# B&R Automation Studio project AriesV2 (part 2)

### _X_bgftpclient.c
```c
#include <bur/plc.h>
#include <bur/plctypes.h>
#include <ethernet.h>
#include <ethsock.h>
#include <asstring.h>
#include <brsystem.h>
#include <sys_lib.h>

#include "bgsprintf.h"
#include "bgstatemachine.h"
#include "bgstring.h"
#include "bgFtpClient.h"

#include "bgdebug.h"

#include "bgstatemachine.c"
#include "bgsprintf.c"
#include "bgstring.c"

/*
History:
9/11/2005
- added support for receiving large files over ftp
- added error event for user ftp commands:
int bgFtpClientCmd<CmdName>OnError(bgFtpClient_typ *p);

*/

void ftpClientConnect(bgFtpClient_typ *p, int msgId);
int ftpClientConnectOnDone(bgFtpClient_typ *p);
int ftpClientConnectOnError(bgFtpClient_typ *p);

void ftpClientLogin(bgFtpClient_typ *p, int msgId);
int ftpClientLoginOnDone(bgFtpClient_typ *p);
int ftpClientLoginOnError(bgFtpClient_typ *p);

void ftpClientLogout(bgFtpClient_typ *p, int msgId);
int ftpClientLogoutOnDone(bgFtpClient_typ *p);
int ftpClientLogoutOnError(bgFtpClient_typ *p);

void ftpClientCmdGetFile(bgFtpClient_typ *p);

void ftpClientCmdList(bgFtpClient_typ *p);

void ftpClientCmdPwd(bgFtpClient_typ *p);

void ftpClientCmdCwd(bgFtpClient_typ *p);

void ftpClientDataServer(bgFtpClient_typ *p, int msgId);
int ftpClientDataServerOnError(bgFtpClient_typ *p);
int ftpClientDataServerOnDone(bgFtpClient_typ *p);

void ftpClientSingleCmdInit(bgFtpClient_typ *p, char *cmd, char *expectedServerResponse);
void ftpClientSingleCmd(bgFtpClient_typ *p);
int ftpClientSingleCmdOnError(bgFtpClient_typ *p);
int ftpClientSingleCmdOnDone(bgFtpClient_typ *p);

void ftpClientExecuteUserCmd_cyclic(bgFtpClient_typ *p);

int ftpClientCmdMultiOnDone(bgFtpClient_typ *p, int cmdId);
int ftpClientMultiCmdOnError(bgFtpClient_typ *p, int cmdId);
int ftpClientCmdCheckServerResponseCode(bgFtpClient_typ *p);

void ftpClientInitDataPort(bgFtpClient_typ *p);
void swapBytesInShort(unsigned short *value);
void setSocketAddressData(ETH_sockaddr_typ *adrData, char *hostIpAddressString, unsigned short hostPort);
void ftpClientGetResponse(bgFtpClient_typ *p);

void ftpClientCmdTextPort(bgFtpClient_typ *p, char *textBuffer);
void ftpClientMutliStateCmdErrorLog(bgFtpClient_typ *p);

int ftpClientIncrDataPort(bgFtpClient_typ *p);

/*
########################################################################################
========================================================================================
- FTP client protocol main state machine
- must be executed as a cyclic task (<=100ms)
- protocol implemenation uses nested state machines (several levels deep)
- FTP functions such as: connect, disconnect, login, logout and different FTP commands
are all implemented as state machines
*/
void bgFtpClientCyclic(bgFtpClient_typ *p, int msgId)
{
bgStateMachine_typ *psm = &p->smFtp;

	/*FTP client top level state machine*/
	switch( bgSMCyclic(psm) ){
		case 1:
          	/*idle; monitor user connection request flag*/
			bgSMSetStateName(psm, "Idle");

          	if(p->user.connectRequest){
	            p->user.connectRequest = 0;
	            p->user.disconnectRequest = 0;
				bgSMSetNextState(psm, bgSMGetState(psm) + 1);
          	}
		break;
		case 2:
			/*connect to FTP server*/
			bgSMSetStateName(psm, "Connect");

			if(bgSMIsStateInit(psm)){
				ftpClientConnect(p, BGSM_MSGID_INIT);
			}

			ftpClientConnect(p, BGSM_MSGID_CYCLIC);

			/*check if we are connected to FTP server*/
			if( p->isConnected ){
				bgSMSetNextState(psm, bgSMGetState(psm) + 1);
			}

			if(	ftpClientConnectOnError(p)){
                ERRxwarning(USER_ERROR_FTP, 1, "ftpClient-Err-socket()");
				bgSMRaiseError(psm, "error in lower level SM", 1, 0);
            }
		break;
		case 3:
			/*login*/
			bgSMSetStateName(psm, "Login");

			if(bgSMIsStateInit(psm)){
				ftpClientLogin(p, BGSM_MSGID_INIT);
			}

			ftpClientLogin(p, BGSM_MSGID_CYCLIC);

			/*check if we are looged-in*/
			if(p->isLoggedIn){
				p->userState = 0;
				bgSMSetNextState(psm, bgSMGetState(psm) + 1);
			}
			if(ftpClientLoginOnError(p)){
                ERRxwarning(USER_ERROR_FTP, 1, "ftpClient-Err-login()");
				bgSMRaiseError(psm, "error in lower level SM", 0, 0);
            }
		break;
		case 4:
            /*connected & logged-in -> normal operational state*/
			bgSMSetStateName(psm, "Ready");

			/*monitor requests & execute FTP commands*/
			ftpClientExecuteUserCmd_cyclic(p);

			/*terminate if socket error detected*/
			if(p->cmdError == ERR_SOCKET){
				bgSMSetNextState(psm, bgSMGetState(psm) + 1);
			}

			if(p->test){
				p->test = 0;
				ftpClientGetResponse(p);
			}

            /*monitor user disconnect request*/
            /*NOTE: upon receiving request, make sure to wait that FTP command in progress completes!*/

			/*disconnect allowed only after command completes*/
            if(p->user.disconnectRequest && !p->userState){
                p->user.connectRequest = 0;
                p->user.disconnectRequest = 0;
				bgSMSetNextState(psm, bgSMGetState(psm) + 1);
            }
		break;
		case 5:
            /*logout*/
			bgSMSetStateName(psm, "Logout");

			if(bgSMIsStateInit(psm)){
				ftpClientLogout(p, BGSM_MSGID_INIT);
			}

			ftpClientLogout(p, BGSM_MSGID_CYCLIC);

			/*chech if we are logged out*/
			if(!p->isLoggedIn){
				bgSMSetNextState(psm, bgSMGetState(psm) + 1);
			}

			if(ftpClientLogoutOnError(p)){
                ERRxwarning(USER_ERROR_FTP, 1, "ftpClient-Err-socket()");
				bgSMRaiseError(psm, "error in lower level SM", 0, 0);
            }
		break;
		case 6:
			bgSMSetStateName(psm, "Close CMD socket");
            /*normal operation; close socket*/
			bgSMRaiseDone(psm, 0);
		break;
		default:
			/*unhandled state*/
			bgSMRaiseError(psm, "unknown state", 0, bgSMGetState(psm));
		break;
	}

	if(bgSMOnDone(psm)){
		/*error state; socket closing is needed*/
		close(p->sock);

		p->isConnected = 0;

		bgSMSetNextState(psm, 1);
	}

	if(bgSMOnError(psm)){
		/*check if socket close needed or not?*/
		if( !bgSMGetErrorId(psm) )
			close(p->sock);

		p->isConnected = 0;
		p->cmdError = 1;
		bgSMSetNextState(psm, 1);
	}
}
/*
########################################################################################
	 INDIVIDUAL FTP COMMANDS
- each individual FTP command has following USER level interface methods:
	ftpClientCmd<Name>Init()
		- start command execution; pass-in user parameters; init cmd state machine
	ftpClientCmd<Name>OnDone()
		- monitor cmd completion (0-not complete; 1-complete)

- each command also has core implemenation (not used or called by the user)
	ftpClientCmd<Name>()

- FTP commands such as: PWD, CWD, PUT, GET, DIR are multi-level commands: it usually takes
several primitive FTP commands (i.e. PORT, TYPE, RETR etc) to complete one FTP command

########################################################################################
*/

/*
========================================================================================
- state machine that handles execution of individual, multi-level FTP commands
- FTP client executes one Multi-level command at the time
*/
void ftpClientExecuteUserCmd_cyclic(bgFtpClient_typ *p)
{
	/*execute user commands*/
	switch(p->userState){
	/*idle*/
        case 0:
        break;
        case 1:
        break;
        case 2:
            ftpClientCmdList(p);
        break;
        case 4:
            ftpClientCmdPwd(p);
        break;
        case 6:
            ftpClientCmdGetFile(p);
        break;
        case 8:
            ftpClientCmdCwd(p);
        break;
        default:
            p->userState = 0;
        break;
	}

}

/*
========================================================================================
FTP Command Implementation:
GetFile
*/
void bgFtpClientCmdGetFileInit(bgFtpClient_typ *p, char *fileName, char* buffer, int bufferLength)
{
    /*select command to execute*/
	p->userState = 6;

	/*pass command parameters*/
	p->user.dataBuffer = buffer;
	p->user.dataBufferLength = bufferLength;
	strcpy(&p->user.fileName[0], fileName);

    /*start command execution*/
	bgSMReset(&p->smFtpMultiCmd);
}

int bgFtpClientCmdGetFileOnDone(bgFtpClient_typ *p)
{
	return ftpClientCmdMultiOnDone(p, 6);
}

int bgFtpClientCmdGetFileOnError(bgFtpClient_typ *p)
{
	return ftpClientMultiCmdOnError(p, 6);
}

void ftpClientCmdGetFile(bgFtpClient_typ *p)
{
char cmdText[256];
bgStateMachine_typ *psm = &p->smFtpMultiCmd;

	/*FTP client multi level command state machine*/
	switch( bgSMCyclic(psm) ){
		case 1:
          	/*idle - monitor user connection request flag*/
			bgSMSetStateName(psm, "GetFile-InitDataSocket");

			if( bgSMIsStateInit(psm) ){
				/*generate port number to use*/
				ftpClientIncrDataPort(p);
				/*init Data transport socket*/
	            ftpClientDataServer(p, BGSM_MSGID_INIT);
			}

			/*wait for ready msg from the DataServer*/
            if( p->isDataPortReady ){
				bgSMSetNextState(psm, bgSMGetState(psm) + 1);
            }
/*TODO: timeout*/
		break;
		case 2:
    		/*PORT command: "PORT 192,168,1,6,0,20<CR><LF>"*/
			bgSMSetStateName(psm, "GetFile-PORT");
			if(bgSMIsStateInit(psm)){
	    		/*send command*/
	            ftpClientCmdTextPort(p, &cmdText[0]);

	    		ftpClientSingleCmdInit(p, &cmdText[0], "2??");
			}

    		/*recv cmd response*/
    		ftpClientSingleCmd(p);
			if(ftpClientSingleCmdOnDone(p)){
				bgSMSetNextState(psm, bgSMGetState(psm) + 1);
			}
			if(ftpClientSingleCmdOnError(p)){
				bgSMRaiseError(psm, "error in lower level SM", 0, 0);
			}
		break;
		case 3:
    		/*TYPE command: "TYPE I<CR><LF>"*/
			bgSMSetStateName(psm, "GetFile-TYPE");
			if(bgSMIsStateInit(psm)){
	    		/*send command*/
	    		ftpClientSingleCmdInit(p, "TYPE I", "2??");
			}

    		/*recv cmd response*/
    		ftpClientSingleCmd(p);
			if(ftpClientSingleCmdOnDone(p)){
				bgSMSetNextState(psm, bgSMGetState(psm) + 1);
			}

			if(ftpClientSingleCmdOnError(p)){
				bgSMRaiseError(psm, "error in lower level SM", 0, 0);
			}
		break;
		case 4:
    		/*RETR command: "RETR<CR><LF>""*/
			bgSMSetStateName(psm, "GetFile-RETR");
			if(bgSMIsStateInit(psm)){
	    		/*send command*/
	    		/*send command*/
	    		strcpy(&cmdText[0], "RETR ");
	    		strcat(&cmdText[0], &p->user.fileName[0]);
	    		ftpClientSingleCmdInit(p, &cmdText[0], "2??");
			}

    		/*recv cmd response*/
    		ftpClientSingleCmd(p);
			if(ftpClientSingleCmdOnDone(p)){
				/*notify data port server that the response is comming*/
				ftpClientDataServer(p, 2);
				bgSMSetNextState(psm, bgSMGetState(psm) + 1);
			}

			if(ftpClientSingleCmdOnError(p)){
				bgSMRaiseError(psm, "error in lower level SM", 0, 0);
				/*close data server port*/
				ftpClientDataServer(p, 3);
			}
		break;
        case 5:
			bgSMSetStateName(psm, "GetFile-DATASRVR active");
        break;
		default:
			/*unhandled state*/
			bgSMRaiseError(psm, "unknown state", 0, bgSMGetState(psm));
		break;
	}

	if(bgSMOnError(psm)){
		p->isErrorMultiCmd = p->userState;
		p->userState = 0;
		return;
	}

	ftpClientDataServer(p, BGSM_MSGID_CYCLIC);

	if(ftpClientDataServerOnDone(p)){
		p->isDoneMultiCmd = p->userState;
		p->userState = 0;
	}

	if(ftpClientDataServerOnError(p)){
		p->isErrorMultiCmd = p->userState;
		p->userState = 0;
	}

}
/*
========================================================================================
FTP Command Implementation:
List (dir)
*/
void bgFtpClientCmdListInit(bgFtpClient_typ *p, char *buffer, int bufferLength)
{
    /*select command to execute*/
	p->userState = 2;

	/*pass command parameters*/
	p->user.dataBuffer = buffer;
	p->user.dataBufferLength = bufferLength;

    /*start command execution*/
	bgSMReset(&p->smFtpMultiCmd);
}

int bgFtpClientCmdListOnDone(bgFtpClient_typ *p)
{
	return ftpClientCmdMultiOnDone(p, 2);
}

int bgFtpClientCmdListOnError(bgFtpClient_typ *p)
{
	return ftpClientMultiCmdOnError(p, 2);

}

void ftpClientCmdList(bgFtpClient_typ *p)
{
char cmdText[64];
bgStateMachine_typ *psm = &p->smFtpMultiCmd;

	/*FTP client multi level command state machine*/
	switch( bgSMCyclic(psm) ){
		case 1:
          	/*idle - monitor user connection request flag*/
			bgSMSetStateName(psm, "List-InitDataSocket");

			if( bgSMIsStateInit(psm) ){
				/*generate port number to use*/
				ftpClientIncrDataPort(p);
				/*init Data transport socket*/
	            ftpClientDataServer(p, BGSM_MSGID_INIT);
			}

			/*wait for ready msg from the DataServer*/
            if( p->isDataPortReady ){
				bgSMSetNextState(psm, bgSMGetState(psm) + 1);
            }
/*TODO: timeout*/
		break;
		case 2:
    		/*PORT command: "PORT 192,168,1,6,0,20<CR><LF>"*/
			bgSMSetStateName(psm, "List-PORT");
			if(bgSMIsStateInit(psm)){
	    		/*send command*/
	            ftpClientCmdTextPort(p, &cmdText[0]);

	    		ftpClientSingleCmdInit(p, &cmdText[0], "2??");
			}

    		/*recv cmd response*/
    		ftpClientSingleCmd(p);
			if(ftpClientSingleCmdOnDone(p)){
				bgSMSetNextState(psm, bgSMGetState(psm) + 1);
			}
			if(ftpClientSingleCmdOnError(p)){
				bgSMRaiseError(psm, "error in lower level SM", 0, 0);
			}
		break;
		case 3:
    		/*TYPE command: "TYPE I<CR><LF>"*/
			bgSMSetStateName(psm, "List-TYPE");
			if(bgSMIsStateInit(psm)){
	    		/*send command*/
	    		ftpClientSingleCmdInit(p, "TYPE I", "2??");
			}

    		/*recv cmd response*/
    		ftpClientSingleCmd(p);
			if(ftpClientSingleCmdOnDone(p)){
				bgSMSetNextState(psm, bgSMGetState(psm) + 1);
			}

			if(ftpClientSingleCmdOnError(p)){
				bgSMRaiseError(psm, "error in lower level SM", 0, 0);
			}
		break;
		case 4:
    		/*LIST command: "LIST<CR><LF>""*/
			bgSMSetStateName(psm, "List-List");
			if(bgSMIsStateInit(psm)){
	    		/*send command*/
	    		ftpClientSingleCmdInit(p, "LIST", "2??");
			}

    		/*recv cmd response*/
    		ftpClientSingleCmd(p);
			if(ftpClientSingleCmdOnDone(p)){
				/*notify data port server that the response is comming*/
				ftpClientDataServer(p, 2);
				bgSMSetNextState(psm, bgSMGetState(psm) + 1);
			}

			if(ftpClientSingleCmdOnError(p)){
				/*close data server port*/
				ftpClientDataServer(p, 3);
				bgSMRaiseError(psm, "error in lower level SM", 0, 0);
			}
		break;
        case 5:
			bgSMSetStateName(psm, "List-DATASRVR active");
        break;
		default:
			/*unhandled state*/
			bgSMRaiseError(psm, "unknown state", 0, bgSMGetState(psm));
		break;
	}

	if(bgSMOnError(psm)){
		p->isErrorMultiCmd = p->userState;
		p->userState = 0;
		return;
	}

	ftpClientDataServer(p, BGSM_MSGID_CYCLIC);

	if(ftpClientDataServerOnDone(p)){
		p->isDoneMultiCmd = p->userState;
		p->userState = 0;
	}

	if(ftpClientDataServerOnError(p)){
		p->isErrorMultiCmd = p->userState;
		p->userState = 0;
	}
}
/*
========================================================================================
FTP Command Implementation:
Pwd (Print Working Directory)
*/
void bgFtpClientCmdPwdInit(bgFtpClient_typ *p, char *buffer, int bufferLength)
{
    /*select command to execute*/
	p->userState = 4;

	/*pass command parameters*/
	p->user.dataBuffer = buffer;
	p->user.dataBufferLength = bufferLength;

    /*start command execution*/
	bgSMReset(&p->smFtpMultiCmd);
}

int bgFtpClientCmdPwdOnDone(bgFtpClient_typ *p)
{
	return ftpClientCmdMultiOnDone(p, 4);
}

int bgFtpClientCmdPwdOnError(bgFtpClient_typ *p)
{
	return ftpClientMultiCmdOnError(p, 4);

}

void ftpClientCmdPwd(bgFtpClient_typ *p)
{
bgStateMachine_typ *psm = &p->smFtpMultiCmd;

	/*FTP client multi level command state machine*/
	switch( bgSMCyclic(psm) ){
		case 1:
    		/*XPWD command: "XPWD<CR><LF>"*/
			bgSMSetStateName(psm, "PWD");
			if(bgSMIsStateInit(psm)){
	    		/*send command*/
	    		ftpClientSingleCmdInit(p, "PWD", "2??");
			}

    		/*recv cmd response*/
    		ftpClientSingleCmd(p);

			if(ftpClientSingleCmdOnDone(p)){
				/*copy response strig into the user supplied buffer*/
				strcpy(p->user.dataBuffer, p->responseList.items[0]);
				bgSMRaiseDone(psm, 0);
			}

			if(ftpClientSingleCmdOnError(p)){
				bgSMRaiseError(psm, "got lower SM error", 0, 0);
			}
		break;
		default:
			/*unhandled state*/
			bgSMRaiseError(psm, "unknown state", 0, bgSMGetState(psm));
		break;
	}

	if(bgSMOnError(psm)){
		p->userState = 0;
	}

	if(bgSMOnDone(psm)){
		p->isDoneMultiCmd = p->userState;
		p->userState = 0;
	}

}
/*
========================================================================================
FTP Command Implementation:
Cwd (Change Working Directory)
*/
void bgFtpClientCmdCwdInit(bgFtpClient_typ *p, char *fileName, char *buffer, int bufferLength)
{
    /*select command to execute*/
	p->userState = 8;

	/*pass command parameters*/
	p->user.dataBuffer = buffer;
	p->user.dataBufferLength = bufferLength;
	strcpy(&p->user.fileName[0], fileName);

    /*start command execution*/
	bgSMReset(&p->smFtpMultiCmd);

}

int bgFtpClientCmdCwdOnDone(bgFtpClient_typ *p)
{
	return ftpClientCmdMultiOnDone(p, 8);
}

int bgFtpClientCmdCwdOnError(bgFtpClient_typ *p)
{
	return ftpClientMultiCmdOnError(p, 8);

}

void ftpClientCmdCwd(bgFtpClient_typ *p)
{
char cmdText[255];

bgStateMachine_typ *psm = &p->smFtpMultiCmd;

	/*FTP client multi level command state machine*/
	switch( bgSMCyclic(psm) ){
		case 1:
    		/*XPWD command: "CWD <fileName><CR><LF>"*/
			bgSMSetStateName(psm, "CWD");
			if(bgSMIsStateInit(psm)){
	    		/*send command: "CWD <fileName><CR><LF>"*/
	    		strcpy(&cmdText[0], "CWD ");
	    		strcat(&cmdText[0], &p->user.fileName[0]);
	    		ftpClientSingleCmdInit(p, &cmdText[0], "2??");
			}

    		/*recv cmd response*/
    		ftpClientSingleCmd(p);

			if(ftpClientSingleCmdOnDone(p)){
				/*copy response strig into the user supplied buffer*/
				strcpy(p->user.dataBuffer, p->responseList.items[0]);
				bgSMRaiseDone(psm, 0);
			}

			if(ftpClientSingleCmdOnError(p)){
				bgSMRaiseError(psm, "got lower SM error", 0, 0);
			}
		break;
	}

	if(bgSMOnError(psm)){
		p->isErrorMultiCmd = p->userState;
		p->userState = 0;
		return;
	}

	if(bgSMOnDone(psm)){
		p->isDoneMultiCmd = p->userState;
		p->userState = 0;
	}
}
/*
########################################################################################
========================================================================================
FTP Connect command state machine:
*/
int ftpClientConnectOnDone(bgFtpClient_typ *p){
	return bgSMOnDone(&p->smCmdSocket);
}

int ftpClientConnectOnError(bgFtpClient_typ *p){
	return bgSMOnError(&p->smCmdSocket);
}

void ftpClientConnect(bgFtpClient_typ *p, int msgId)
{
DINT ret;
bgStateMachine_typ *psm = & p->smCmdSocket;

	if( msgId == BGSM_MSGID_INIT){
		bgSMReset(psm);
	}

    switch(bgSMCyclic(psm)){
        case 1:
			bgSMSetStateName(psm, "Connect-CreateSocket");

			if( bgSMIsStateInit(psm) ){
				p->cmdError = 0;
				p->cmdErrorCode = 0;
				p->isConnected = 0;
				/*create socket*/
				p->sock = socket(ETH_AF_INET, ETH_SOCK_STREAM, 0);

				if( p->sock == ERR_SOCKET ){
					bgSMRaiseError(psm, "socket create err", 0, EthGetError());
					break;
				}

				/*set non-blocking socket operation*/
				{
					UDINT arg = 1;
					ioctl(p->sock, ETH_FIONBIO, (UDINT)&arg);
				}

				/*reset select flags*/
				fd_zero((UDINT)&p->fdR);
				fd_zero((UDINT)&p->fdW);

				/*set time-out to 10ms*/
				p->timeOut.tv_sec = 0;
				p->timeOut.tv_usec = 1000 * 10;

				/*adjust my own timeout counters*/
				p->sockData_TimerCounter = 0;
				p->sockData_TimerTime = 10;
#if 0
/*bind not necessary*/
				/*bind client socket*/
				ret = bind(p->sock, (UDINT)&p->ftpClientAdrData, sizeof(p->ftpClientAdrData));
				if(ret == ERR_SOCKET){
					bgSMRaiseError(psm, "socket bind err", 0, EthGetError());
					break;
				}
#endif
			}

			/*connect to remote host*/
			ret = connect(p->sock, (UDINT)&p->ftpServerAdrCmd, sizeof(p->ftpServerAdrCmd) );

			if(ret == ERR_SOCKET){
				UINT errCode = EthGetError();
				if(errCode == ERR_ETH_INPROGRESS){
					/*next: wait connect to complete*/
					bgSMSetNextState(psm, bgSMGetState(psm) + 1);
				    break;
				}else
				if(errCode == ERR_ETH_ISCONN){
					/*it's connected -> done*/
					ERRxwarning(USER_ERROR_FTP, errCode, "connect()-alreadyOK!");
					bgSMRaiseDone(psm, 0);
					break;
				}
				else{
					bgSMRaiseError(psm, "socket connect err", 0, EthGetError());
					break;
				}
			}
			/*connected!*/
			ERRxwarning(USER_ERROR_FTP, ret, "connect()-OK-Quick!");
			bgSMRaiseDone(psm, 0);
		break;
		case 2:
			bgSMSetStateName(psm, "Connect-Connect");

			/*select waits for connection to complete*/
			fd_set(p->sock, (UDINT)&p->fdR);
			fd_set(p->sock, (UDINT)&p->fdW);
			ret = sock_select(32, (UDINT)&p->fdR, (UDINT)&p->fdW, 0L, (UDINT)&p->timeOut);

			if(ret == ERR_SOCKET){
				bgSMRaiseError(psm, "socket connect err", 0, EthGetError());
				break;
			}
/*
			DBG("connect: ret=%d, error=%d\n\r", ret, EthGetError());
*/
			if(ret == 0){
				if( p->sockData_TimerCounter >= p->sockData_TimerTime ){
					/*NOTES:
					- trying to figure out how does the select timeout works in B&R!
					- using EthGetError() here is not needed, just to see what comes back
					*/
					bgSMRaiseError(psm, "connect timeout", 0, EthGetError());
				}else{
					p->sockData_TimerCounter++;
				}
			}else{
				if( fd_isset(p->sock, (UDINT)&p->fdW) ){
					bgSMRaiseDone(psm, 0);
				}
			}
		break;
		default:
			/*unhandled state*/
			bgSMRaiseError(psm, "unknown state", 0, bgSMGetState(psm));
		break;
    }

	if( bgSMOnDone(psm)){
		ERRxwarning(USER_ERROR_FTP, 0, "connect()-OK!");
		p->isConnected = 1;
	}

	if( bgSMOnError(psm)){

	}
}
/*
========================================================================================
*/
void ftpClientMutliStateCmdErrorLog(bgFtpClient_typ *p){
char text[64];
	/*log error*/
	strcpy(&text[0], "Err: ");
	strcat(&text[0], &p->cmdSendBuf[0]);
    ERRxwarning(USER_ERROR_FTP, p->cmdErrorCode, &text[0]);
}
/*
########################################################################################
========================================================================================
FTP Login command state machine:
-return values:
*/
int ftpClientLoginOnDone(bgFtpClient_typ *p){
	return bgSMOnDone(&p->smFtpMultiCmd);
}

int ftpClientLoginOnError(bgFtpClient_typ *p){
	return bgSMOnError(&p->smFtpMultiCmd);
}
void ftpClientLogin(bgFtpClient_typ *p, int msgId)
{
bgStateMachine_typ *psm = &p->smFtpMultiCmd;

	if( msgId == BGSM_MSGID_INIT){
		bgSMReset(psm);
	}

    switch(bgSMCyclic(psm)){
        case 1:
			/*send USER name*/
			bgSMSetStateName(psm, "Login-Welcome");

			if( bgSMIsStateInit(psm) ){
				/*send request*/
				/*ftpClientSingleCmdInit(p, 0, ">name");*/
				ftpClientSingleCmdInit(p, 0, ">FTP");
			}

			/*recv response*/
			ftpClientSingleCmd(p);

			if(ftpClientSingleCmdOnDone(p)){
				bgSMSetNextState(psm, bgSMGetState(psm) + 1);
			}

			if(ftpClientSingleCmdOnError(p)){
				bgSMRaiseError(psm, "error in lower level SM", 0, 0);
			}
        break;
        case 2:
			/*send USER name*/
			bgSMSetStateName(psm, "Login-UserName");

			if( bgSMIsStateInit(psm) ){
				/*send request*/
				ftpClientSingleCmdInit(p, "USER  anonymous", "331");
			}

			/*recv response*/
			ftpClientSingleCmd(p);

			if(ftpClientSingleCmdOnDone(p)){
				bgSMSetNextState(psm, bgSMGetState(psm) + 1);
			}

			if(ftpClientSingleCmdOnError(p)){
				bgSMRaiseError(psm, "error in lower level SM", 0, 0);
			}
        break;
        case 3:
			/*send PASSWORD */
			bgSMSetStateName(psm, "Login-Password");

			if( bgSMIsStateInit(psm) ){
				/*send request*/
				ftpClientSingleCmdInit(p, "PASS  anonymous@", "230");
			}

			/*recv response*/
			ftpClientSingleCmd(p);

			if(ftpClientSingleCmdOnDone(p)){
				bgSMRaiseDone(psm, 0);
			}

			if(ftpClientSingleCmdOnError(p)){
				bgSMRaiseError(psm, "error in lower level SM", 0, 0);
			}
        break;
        default:
			/*unhandled state*/
			bgSMRaiseError(psm, "unknown state", 0, bgSMGetState(psm));
        break;
    }

	if( bgSMOnDone(psm) ){
		p->isLoggedIn = 1;
	}

	if( bgSMOnError(psm) ){
		ftpClientMutliStateCmdErrorLog(p);
	}

}
/*
########################################################################################
========================================================================================
FTP Logout command state machine:
-return values:
*/
int ftpClientLogoutOnDone(bgFtpClient_typ *p){
	return bgSMOnDone(&p->smFtpMultiCmd);
}

int ftpClientLogoutOnError(bgFtpClient_typ *p){
	return bgSMOnError(&p->smFtpMultiCmd);
}

void ftpClientLogout(bgFtpClient_typ *p, int msgId)
{
bgStateMachine_typ *psm = &p->smFtpMultiCmd;

	if( msgId == BGSM_MSGID_INIT){
		bgSMReset(psm);
	}

    switch(bgSMCyclic(psm)){
        case 1:
			/*send USER name*/
			bgSMSetStateName(psm, "Logout-Quit");

			if( bgSMIsStateInit(psm) ){
				/*send request*/
				ftpClientSingleCmdInit(p, "QUIT", "2??");
			}

			/*recv response*/
			ftpClientSingleCmd(p);

			if(ftpClientSingleCmdOnDone(p)){
				bgSMRaiseDone(psm, 0);
			}

			if(ftpClientSingleCmdOnError(p)){
				bgSMRaiseError(psm, "error in lower level SM", 0, 0);
			}
        break;
        default:
			/*unhandled state*/
			bgSMRaiseError(psm, "unknown state", 0, bgSMGetState(psm));
        break;
    }

	if(bgSMOnDone(psm)){
		p->isLoggedIn = 0;
	}

	if(bgSMOnError(psm)){
		p->isLoggedIn = 0;
		ftpClientMutliStateCmdErrorLog(p);
	}
}
/*
########################################################################################
========================================================================================
Lowest level state machine handles execution of a single FTP request/response messaging

ftpClientSingleCmdInit();
	- selects command to execute; init command state machine

ftpClientSingleCmd();
	- command execution state machine

ftpClientCmdCheckServerResponseCode()
	- command response check and verification

*/
void ftpClientSingleCmdInit(bgFtpClient_typ *p, char *cmd, char *expectedServerResponse){
int i;

	/*copy command string into send buffer*/
	p->cmdSendBuf[0]=0;
	if(cmd){
		strcpy(&p->cmdSendBuf[0], cmd);
		/*append string termination -> CRLF*/
		strcat(&p->cmdSendBuf[0], "\r\n");
	}

	/*define expected server response string?*/
	p->cmdExpectedServerResponse[0] = 0;	/*don't care*/
	if(expectedServerResponse){
		/*is expected server response code or string?*/
		if( *expectedServerResponse == '>'){
			i = 1;
			p->cmdExpectedServerResponseCodeOrString = 1;	/*string*/
		}else{
			i = 0;
			p->cmdExpectedServerResponseCodeOrString = 0;	/*code*/
		}
		bgStrCpyN(&p->cmdExpectedServerResponse[0], expectedServerResponse+i, FTPCLIENT_RESPONSECODE_LEN);
	}

	/*clr rcv buffer string*/
	memset(&p->cmdRecvBuf[0], 0, FTPCLIENT_CMDBUFSIZE);
#if 0
/*clear response lines*/
	/*init ptrs*/
	p->responseList.maxCount = CMD_RESPONSE_MAXLINES;
	p->responseList.lines[0] = &p->responseList.line0[0];
	p->responseList.lines[1] = &p->responseList.line1[0];
	p->responseList.lines[2] = &p->responseList.line2[0];
	p->responseList.lines[3] = &p->responseList.line3[0];
	p->responseList.lines[4] = &p->responseList.line4[0];

	/*clear all response lines*/
	for(i=0;i<CMD_RESPONSE_MAXLINES; i++){
		memset(p->responseList.lines[i], 0, CMD_RESPONSE_MAXLINELEN);
	}
	/*number of lines retrieved from the cmd buffer*/
	p->responseList.count = 0;
#endif
	/*number of lines retrieved from the cmd buffer*/
	p->responseList.itemCount = 0;

	/*reset command execution state machine*/
	bgSMReset(&p->smFtpCmd);
}

void ftpClientSingleCmd(bgFtpClient_typ *p){
DINT len;
DINT ret;
bgStateMachine_typ *psm = &p->smFtpCmd;

	/*state machine states*/
	switch( bgSMCyclic(psm) ){
		case 1:
          	/*send command request*/
			bgSMSetStateName(psm, "ftpSingleCmd");

			if(bgSMIsStateInit(psm)){
				/*check input conditions and paramters*/
				if( !p->isConnected ){
					bgSMRaiseError(psm, "not connected", 0, 0);
					break;
				}
				if( !p->cmdSendBuf[0]){
					/*nothing to send! receive only (i.e. welcome message just after connect()*/
					break;
				}

				/*send command to server*/
	         	len = strlen(&p->cmdSendBuf[0]);
	        	ret = send(p->sock, (UDINT)&p->cmdSendBuf[0], len, 0L);

	        	if(ret == ERR_SOCKET){
					bgSMRaiseError(psm, "send() error", 0, EthGetError());
					break;
	        	}

				/*remember the send length*/
				DBG("Single CMD send();Bytes=%d;[%s]\r\n", (int)ret, &p->cmdSendBuf[0]);
				p->sendLen = ret;
				return;
			}

	       	/*call receive (NON BLOCKING MODE!)*/
        	ret = recv(p->sock, (UDINT)&p->cmdRecvBuf[0],  FTPCLIENT_CMDBUFSIZE, 0L);

        	if(ret == ERR_SOCKET){
        		UINT errCode = EthGetError();
        		/*none blocking receive return this following value if data is not available yet*/
        		if( errCode == ERR_ETH_WOULDBLOCK ){
        			/*wait response*/
					return;
        		}

				/*recv error*/
				bgSMRaiseError(psm, "recv() error", 0, EthGetError());
				break;
        	}

			if(ret == 0){
				bgSMRaiseError(psm, "rx len=0", 0, 0);
				return;
			}

			/*receive is complete; store receive length & terminate rx buffer*/
			p->cmdRecvBuf[ret] = 0;
			DBG("Single CMD recv();Bytes=%d;[%s]\r\n", (int)ret, &p->cmdRecvBuf[0]);
			p->recvLen = ret;

			ret = ftpClientCmdCheckServerResponseCode(p);

			if( ret == 1)
				bgSMRaiseDone(psm, 0);

			if( ret == 2)
				bgSMRaiseError(psm, "server error response", 0, 0);

		break;
		default:
			/*unhandled state*/
			bgSMRaiseError(psm, "unknown state", 0, bgSMGetState(psm));
		break;
	}

	/*error event handler*/
	if(bgSMOnError(psm)){
		DBG("ftpClientSingleCmd - ERROR.\r\n");
	}

	/*done event handler*/
	if(bgSMOnDone(psm)){
		DBG("ftpClientSingleCmd - DONE.\r\n");
	}
}

int ftpClientSingleCmdOnError(bgFtpClient_typ *p)
{
	return bgSMOnError(&p->smFtpCmd);
}

int ftpClientSingleCmdOnDone(bgFtpClient_typ *p)
{
	return bgSMOnDone(&p->smFtpCmd);
}

/*
========================================================================================
FTP command response code is an ASCII line that looks like:
"xyz-response text<CR><LF>"
where x,y,z are numeric chars <0-9> followed by a '-' and the response text
- multiple lines per response are possible
- this function retrieves the response from the server, formats it into a list (array) of lines
and then searches each line for the user supplied code (res1,res2,res3)
- if res<x> is given as 0, it means don't care (see ftp spec)

*/
int ftpClientCmdCheckServerResponseCode(bgFtpClient_typ *p)
{
char serverResponseCode[3];
char *line;
int result;
int i;

	/*get server's response
	IMPORTANT:
	- note that data for ftpClientGetResponse() method is initilized within ftpClientSingleCmdInit()!
	- order of execution is like:
		init:
			ftpClientSingleCmdInit();
		cyclic:
			if( ftpClientSingleCmd() == DONE )
				if( ftpClientCmdCheckServerResponseCode() == OK )
					nextState;

	- therfore, the ftpClientGetResponse() shall be designed to operate in an incremenal mode: every time
	ftpClientSingleCmd() completes (data is available in the receive buffer) we should just add to the existing lines
	and not delete what we've received till that moment
	*/
	ftpClientGetResponse(p);

	/*final result of the ftpClientCmdCheckServerResponseCode() method:
	0 - response not found (not available -> wait)
	1 - response found (and it's ok; match with expected response)
	2 - response found (and it's not ok; error response from server)
	*/
	p->serverResponseCode = 0;

	/*anything to process!?*/
	if(!p->responseList.itemCount)
		return 0;

	/*check all received response lines every time (not necessary but it's easy to implement and it does not metter*/
	for(i=0; i<p->responseList.itemCount; i++){
		line = p->responseList.items[i];

		if(!p->cmdExpectedServerResponseCodeOrString){
			serverResponseCode[0]=*(line+0);
			serverResponseCode[1]=*(line+1);
			serverResponseCode[2]=*(line+2);

			result = 0;
			if( p->cmdExpectedServerResponse[0] != '?'){
				if(p->cmdExpectedServerResponse[0] == serverResponseCode[0])
					result++;
			}else
				result++;

			if( p->cmdExpectedServerResponse[1] != '?'){
				if(p->cmdExpectedServerResponse[1] == serverResponseCode[1])
					result++;
			}else
				result++;

			if( p->cmdExpectedServerResponse[2] != '?'){
				if(p->cmdExpectedServerResponse[2] == serverResponseCode[2])
					result++;
			}else
				result++;

			if( result >= 3)
				return 1;

			if( (serverResponseCode[0] == '4') || (serverResponseCode[0] == '5'))
				return 2;
		}else{
			result = bgStrFind(line, &p->cmdExpectedServerResponse[0], -1, -1);

			if(result >= 0)
				return 1;
		}
	}

	return 0;
}
/*
========================================================================================
*/
void ftpClientGetResponse(bgFtpClient_typ *p){
int i;
char *src;

	/*ptr to rcv buffer*/
	src = &p->cmdRecvBuf[0];
	p->responseList.src = src;
	bgStringListLines(&p->responseList);

	DBG("Received Cmd Response: lines=%d\r\n", p->responseList.itemCount);
	for(i=0;i<p->responseList.itemCount;i++){
		DBG("Line[%d]=%s\r\n", i, p->responseList.items[i]);
	}

}

int readline(char *src, char *dest, int maxLength){
/*
return: >= 0 (length of the line including CRLF)
return: -1 (no line read)
*/
int lineLen;
char *cPtr;

	lineLen = 0;
	cPtr = src;
	while(maxLength--){

		if( (*cPtr == 0x0D) || ( *cPtr == 0x0A) ){

			lineLen++;
			cPtr++;

			if( (*cPtr == 0x0D) || ( *cPtr == 0x0A) ){
				lineLen++;
			}

			memcpy(dest, src, lineLen);
			*(dest+lineLen+1)= 0;
			return lineLen;
		}

		if( *cPtr == 0 )
			return -1;

		lineLen++;
		cPtr++;
	}

	return -1;
}

/*
========================================================================================
*/
int ftpClientCmdMultiOnDone(bgFtpClient_typ *p, int cmdId)
{
/*generate CmdIsDone signal (1 shoot)*/
	if( p->isDoneMultiCmd == cmdId ){
		p->isDoneMultiCmd = 0;
		return 1;
	}else
		return 0;
}

int ftpClientMultiCmdOnError(bgFtpClient_typ *p, int cmdId){
/*generate CmdIsError signal (1 shoot)*/
	if( p->isErrorMultiCmd == cmdId ){
		p->isErrorMultiCmd = 0;
		return 1;
	}else
		return 0;
}

/*
========================================================================================
*/
void bgFtpClientConnectAndLogin(bgFtpClient_typ *p, char *ethernetDevice, char *serverIp)
{
unsigned long ipAddrClient;

    /*set server ip address and ports to use*/
    /*  21 - standard FTP command port
        20 - standard FTP data port
    */
	setSocketAddressData(&p->ftpServerAdrCmd, serverIp, 21);
	setSocketAddressData(&p->ftpClientAdrData, "", ETH_INADDR_ANY);

	/*retrieve own ip address*/
	p->CfgIPAddr_1.enable = 1;
	p->CfgIPAddr_1.pDevice = (UDINT)ethernetDevice;
	p->CfgIPAddr_1.pIPAddr = (UDINT)&p->CfgIPAddrString[0];
	p->CfgIPAddr_1.Len = 16;
	CfgGetIPAddr(&p->CfgIPAddr_1);

	ipAddrClient = inet_addr( (unsigned long) &p->CfgIPAddrString[0]);

	/*store ip address in an easy format for later use; see PORT command*/
	p->ipAddr[3]= (ipAddrClient>>24)&0xFF;
	p->ipAddr[2]= (ipAddrClient>>16)&0xFF;
	p->ipAddr[1]= (ipAddrClient>>8)&0xFF;
	p->ipAddr[0]= (ipAddrClient)&0xFF;

	p->cmdError = 0;
	p->cmdErrorCode = 0;
	p->isConnected = 0;
    p->user.connectRequest = 1;
}
/*
========================================================================================
*/
int bgFtpClientIsLoggedIn(bgFtpClient_typ *p)
{
    return p->isLoggedIn;
}

/*
========================================================================================
*/
void bgFtpClientDisconnect(bgFtpClient_typ *p)
{
    p->user.disconnectRequest = 1;
}
/*
========================================================================================
*/
int bgFtpClientIsConnected(bgFtpClient_typ *p)
{
    return p->isConnected;
}
/*
========================================================================================
*/
int bgFtpClientIsError(bgFtpClient_typ *p)
{
    return p->cmdError;
}

int ftpClientIncrDataPort(bgFtpClient_typ *p){

	if( !p->dataPort){
		p->dataPort = 190;
	}

	if(p->dataPort>=190)
		p->dataPort++;

	if(p->dataPort>=200)
		p->dataPort = 190;

	return p->dataPort;
}
/*
========================================================================================
*/
void ftpClientCmdTextPort(bgFtpClient_typ *p, char *textBuffer)
{
/*
	bgsprintf(textBuffer, "PORT 192,168,1,6,4,%d", p->dataPort);
*/
	bgsprintf(textBuffer, "PORT %d,%d,%d,%d,4,%d", p->ipAddr[0], p->ipAddr[1], p->ipAddr[2], p->ipAddr[3], p->dataPort);
}
/*
========================================================================================
*/
int ftpClientDataServerOnError(bgFtpClient_typ *p)
{
	return bgSMOnError(&p->smDataSocket);
}

int ftpClientDataServerOnDone(bgFtpClient_typ *p)
{
	return bgSMOnDone(&p->smDataSocket);
}

void ftpClientDataServer(bgFtpClient_typ *p, int msgId)
{
bgStateMachine_typ *psm = &p->smDataSocket;

    /*init data socket (listen)*/
	if( (msgId == BGSM_MSGID_INIT) ){
		bgSMReset(psm);
		p->sockData_TimerTime = 10;
		p->sockData_TimerCounter = 0;
		p->recvLenData = 0;
		p->sendLenData = 0;
		return;
	}

    /*close data socket (listen stop)*/
	if( msgId == 2){
		/*command socket is telling us to receive data from server
		after this event, keep receiving until we don't get any data
		for a certain period of time or the remote host closes the
		connection
		*/
		p->sockData_Timer = 1;
		p->sockData_TimerTime = 20;
		p->sockData_TimerCounter = 0;
		return;
	}

    /*close data socket now!*/
	if( msgId == 3){
		/*command socket is telling us to immediately close data socket
		*/
		bgSMSetNextState(psm, 3);
		return;
	}

	switch(bgSMCyclic(psm)){
		case 1:
			bgSMSetStateName(psm, "DataPort-Init");
			if(bgSMIsStateInit(psm)){
				p->sockData_Timer = 0;

				p->TCPserv_1.enable = 1;            /* enables the FUB */
	    		p->TCPserv_1.porta = 4*256 + p->dataPort;           	/* port number of the server */
	    		TCPserv(&p->TCPserv_1);				/* makes a connection with the clients */

	    		p->TCPrecv_1.enable = 1;           	/* enables the FUB */
				p->rxDataBuff = 0;
				p->recvLenData = 0;
				p->TCPrecv_1.mxbuflng = 10000;		/* size of the buffer should be > 8192*/
    			TMP_alloc (p->TCPrecv_1.mxbuflng, (void**)&p->rxDataBuff);   /*allocate memory for data rx*/
	    		p->TCPrecv_1.buffer = (UDINT)p->rxDataBuff; /* address of the buffer */

	    		p->TCPclose_1.enable = 1;                  /* enables the FUB */

				DBG("data port open\r\n");
				break;

			}

    		TCPserv(&p->TCPserv_1);					/*listen for a server connection request*/

			/*server connection accepted*/
			if(p->TCPserv_1.status == 0){
				/*NOTE: data port is ready if either connection is accepted or if waiting for connection*/
				DBG("datasocket - connected\r\n");
				p->isDataPortReady = 1;
 				bgSMSetNextState(psm, bgSMGetState(psm) + 1);
				break;
			}

			/*waiting for connection || pNA is busy*/
			if( (p->TCPserv_1.status == 0xFFFF) || (p->TCPserv_1.status == 14893) ){
				DBG("datasocket - waiting connection\r\n");
				p->isDataPortReady = 1;
				break;
			}

			DBG("datasocket - error=%d\r\n", p->TCPserv_1.status);

			bgSMRaiseError(psm, "TCPserv() error", 0, p->TCPserv_1.status);
		break;
		case 2:
			bgSMSetStateName(psm, "DataPort-Recv");
			/* recv in progress*/
   			p->TCPrecv_1.cident = p->TCPserv_1.cident;    /* copy serv() Id to recv() */
           	TCPrecv(&p->TCPrecv_1);

			/*recv timer*/
		p->sockData_TimerCounter++;
            if(p->sockData_Timer && (p->TCPrecv_1.status == 0xFFFF)){
    			/*p->sockData_TimerCounter++;*/
				DBG("data port recv() busy; counter=%d\r\n", p->sockData_TimerCounter);
            }

            if(p->TCPrecv_1.status == 0){
				/*test only; inc receive counter*/
				p->counter++;

				/*in case data arrives->copy data to user buffer*/
				if(p->TCPrecv_1.rxbuflng != 0){

					if(p->user.dataBufferLength < (p->recvLenData + p->TCPrecv_1.rxbuflng) ){
						DBG("!!!! rxBufferOverflow rxLen=%d > rxBufferSize=%d!!!!\r\n", (int)(p->recvLenData + p->TCPrecv_1.rxbuflng), (int)p->user.dataBufferLength);
						DBG("!!!! INCREASE USER RX BUFFER SIZE !!!!\r\n");
						/*user supplied buffer is too small!!!*/
						bgSMRaiseError(psm, "Data Buffer Overflow!", 0, bgSMGetState(psm));
						break;
					}

					memcpy( (char*)(p->user.dataBuffer + p->recvLenData), p->rxDataBuff, p->TCPrecv_1.rxbuflng);
					p->recvLenData += p->TCPrecv_1.rxbuflng;

					p->sockData_TimerCounter = 0;
				}
				else{
					/*Status == 0 && rxLengt == 0 -> remote peer has closed the connection!!!*/
					bgSMSetNextState(psm, bgSMGetState(psm) + 1);
				}
            }
			else
			if(p->sockData_TimerCounter >= p->sockData_TimerTime){
				/*if receive timer expires, close data socket*/
				bgSMSetNextState(psm, bgSMGetState(psm) + 1);
			}

			DBG("data recv(); rxLen=%d, rxStatus=%d, timer=%d \r\n",
				(int)p->TCPrecv_1.rxbuflng, (int)p->TCPrecv_1.status, (int)p->sockData_TimerCounter);
		break;
		case 3:
			bgSMSetStateName(psm, "DataPort-Close");
   			p->TCPclose_1.cident = p->TCPserv_1.cident;    	/* copy the  Ident number */
            TCPclose(&p->TCPclose_1);          /* set the socket free */

			if(p->TCPclose_1.status == 0){
				p->isDataPortReady = 0;
				p->sockData_Timer = 0;

				/*terminate rx buffer with 0 -> for strings*/
				p->user.dataBuffer[p->recvLenData] = 0;

				bgSMRaiseDone(psm, 0);
			}

			if( p->rxDataBuff ){
				p->rxDataBuff = 0;
				TMP_free (p->TCPrecv_1.mxbuflng, (void**)p->rxDataBuff);
			}
		break;
		default:
			/*unhandled state*/
			bgSMRaiseError(psm, "unknown state", 0, bgSMGetState(psm));
		break;
	}

	if(bgSMOnError(psm)){
		p->TCPclose_1.cident = p->TCPserv_1.cident;    	/* copy the  Ident number */
	    TCPclose(&p->TCPclose_1);          				/* set the socket free */
		p->isDataPortReady = 0;

		if( p->rxDataBuff ){
			p->rxDataBuff = 0;
			TMP_free (p->TCPrecv_1.mxbuflng, (void**)p->rxDataBuff);
		}
		/*raise error again for cmd level state machine*/
		bgSMRaiseError(psm, "Data Server Error", 0, 0);
 	}

	if(bgSMOnDone(psm)){

	}
}
/*
========================================================================================
*/
void swapBytesInShort(unsigned short *value)
{

union{
	unsigned short 	shortValue;
	unsigned char	bytes[2];
}swapValue;

unsigned char tempByte;

	swapValue.shortValue = *value;
	tempByte = swapValue.bytes[0];
	swapValue.bytes[0] = swapValue.bytes[1];
	swapValue.bytes[1] = tempByte;
	*value = swapValue.shortValue;
}
/*
========================================================================================
*/
void setSocketAddressData(ETH_sockaddr_typ *adrData, char *hostIpAddressString, unsigned short hostPort)
{

	unsigned short sin_family;
	unsigned short family;
	unsigned short length;
	unsigned short port;

	family = ETH_AF_INET;
	length = sizeof(ETH_sockaddr_typ);
	sin_family = (family << 8) + length;

	adrData->sin_family = sin_family;
	port = hostPort;
	swapBytesInShort(&port);
	adrData->sin_port = port;
	if( strlen(hostIpAddressString) < 8)
		adrData->sin_addr = ETH_INADDR_ANY;
	else
		adrData->sin_addr = inet_addr( (unsigned long) hostIpAddressString);
	adrData->sin_zero[0]=0;
	adrData->sin_zero[1]=0;
	adrData->sin_zero[2]=0;
	adrData->sin_zero[3]=0;
	adrData->sin_zero[4]=0;
	adrData->sin_zero[5]=0;
	adrData->sin_zero[6]=0;
	adrData->sin_zero[7]=0;
}
/*
========================================================================================
========================================================================================
========================================================================================
========================================================================================
*/
/*EOF*/
```

### bgfsig.c
```c
#include <bur/plc.h>
#include <bur/plctypes.h>

#include "bglib/bgdebug.h"
#include "bglib/bgstring.h"
#include "bglib/bgSecMD5Signature.h"
#include "bgfsig.h"

/*define a limit for number of lines within a file*/
#define MAX_NUMBER_OF_LINES	3000

static int bgGetLineFromTextBuffer(char* pText, char** pLineNext, char* pDest, int maxLen, int* charCount);

#define  secretWord "NONE!"

/*=============================================================*/
int bgFileSignatureVerify(char *inFileBuffer, char *resultStringMinLen64)
{
int i, index;
char lineBuffer[255];
char lineBufferRaw[255];
int lineCount;
int charCount;
bgStringList_typ splitLine;
md5_state_t state;
md5_byte_t digest[16];
char hexDigestCalculated[40];
char hexDigestFromFile[40];

char *pLineCurrent;
char *pLineNext;

	/*init digest*/
	md5_init(&state);

	/*init hexDigestFromFile as empty*/
	hexDigestFromFile[0] = 0;

	/*init line ptr-s*/
	pLineCurrent = inFileBuffer;
	pLineNext = 0L;

	lineCount = 0;

	/*process all lines from the file*/
	while( 1 ){
	int isNextLinePresent;

		isNextLinePresent = bgGetLineFromTextBuffer(pLineCurrent, &pLineNext, lineBufferRaw, 255, &charCount);

		if( lineCount++ > MAX_NUMBER_OF_LINES){
			DBGCRT("Supplied file buffer has more then %d lines!\r\n", lineCount);
			if( resultStringMinLen64 )
				strcpy(resultStringMinLen64, "Err: file is too long!");
			return -2;
		}

		/*copy a trimmed line into the local buffer*/
		charCount = bgStrCpyNTrimLeadingSpaces(lineBuffer, lineBufferRaw, 255);

		/*check for empty lines & comments*/
		if( !charCount || (lineBuffer[0] == '*')){
			/*empty lines or comments -> skip and go to the next line*/
		}else{
			/*check if this is a signature line*/
			index = bgStrFind(lineBuffer, "SIGNATURE", -1, 0);
			if( index >= 0){
				/*line w. signature -> extract signature stored in the file*/
				splitLine.src = lineBuffer;
				bgStringSplitLine(&splitLine, '=');
				if( splitLine.itemCount != 2){
					DBGCRT("Can't extract signature from the supplied file buffer\r\n");
					if( resultStringMinLen64 )
						strcpy(resultStringMinLen64, "Err: can't extract signature");
					return -2;
				}
				/*copy extracted signature from the file into the local buffer*/
				bgStrCpyN(hexDigestFromFile, splitLine.items[1], 40);
				bgStringUpper(hexDigestFromFile);

			}else{
				/*line wo. signature -> use (append) for digest calculation*/
				md5_append(&state, (const md5_byte_t *)lineBuffer, strlen(lineBuffer));
			}
		}

		/*process next line*/
		if( isNextLinePresent )
			pLineCurrent = pLineNext;
		else
			break;
	}

	/*append secret content*/
	md5_append(&state, (const md5_byte_t *)secretWord, strlen(secretWord));

	/*generate digest*/
	md5_finish(&state, digest);

	/*convert calculated digest into a hex string*/
	for (i = 0; i < 16; ++i)
	    bgsprintf(hexDigestCalculated + i * 2, "%02X", digest[i]);

	/*check if supplied file buffer had stored digital signature*/
	if( !hexDigestFromFile[0] ){
		/*digital signature was NOT present in this file->return result and current (calculated) file digest*/
		if( resultStringMinLen64 )
			bgsprintf(resultStringMinLen64, "StoredSig=NONE CalcSig=%s\n\r", hexDigestCalculated);
		return 0;

	}else{
		/*digital signature IS present in this file->compare calculated and stored signaure*/

		for (i = 0; i < 32; i++){
			if(hexDigestCalculated[i] != hexDigestFromFile[i] ){
				/*digital signatures are not equal -> exit*/
				if( resultStringMinLen64 )
					bgsprintf(resultStringMinLen64, "StoredSig=%s CalcSig=%s\n\r", hexDigestFromFile, hexDigestCalculated);

				return 2;
			}
		}

		/*digital signature verified! stored and calculated signatures are equal!*/
		if( resultStringMinLen64 )
			bgsprintf(resultStringMinLen64, "StoredSigEQUALCalcSig=%s\n\r", hexDigestCalculated);

		return 1;

	}
}
/*=============================================================*/

/*
Input(s):
char *pText - ptr to the text buffer from which to extract a line
char *pDest - destination buffer where to copy the content of a line
int maxLen - max length of the destination buffer

Output(s):
char **pLineNext - ptr to the next line
int *charCount - total number of chars copied into the dest buffer

Return:
0 - there is no more lines in the supplied text buffer
1 - more lines are present in the supplied text buffer
*/
static int bgGetLineFromTextBuffer(char* pText, char** pLineNext, char* pDest, int maxLen, int* charCount)
{

unsigned char *ptrItemStart, *ptrItemEnd;
unsigned char *ptrCpyDest;

	/*init ptrs to the start of the text buffer*/
	ptrItemStart = pText;
	ptrItemEnd = pText;
	ptrCpyDest = pDest;

	/*basic check*/
	if( *ptrItemStart == 0){
		return 0;
	}

	*charCount = 0;
	while( 1 ){
		if( (*ptrItemEnd == 0x0D) || (*ptrItemEnd == 0x0A)){
			/*EOF line char found! -> exit*/
			ptrItemEnd++;

			/*check for an additional \r or \n*/
			if( (*ptrItemEnd == 0x0D) || (*ptrItemEnd == 0x0A)){
				ptrItemEnd++;
			}

			ptrItemStart = ptrItemEnd;

			/*terminate dest buffer*/
			*ptrCpyDest = 0;

			/*check for an end of the text*/
			if( (*ptrItemEnd == 0) ){
				*pLineNext = 0L;
				/*0 -> there are NO more lines in the text buffer*/
				return 0;
			}else{
				*pLineNext = ptrItemStart;
				/*1 -> there are more lines in the text buffer*/
				return 1;
			}
		}else
		if( *ptrItemEnd == 0){
			/*end of text buffer found! -> exit*/

			/*terminate dest buffer*/
			*ptrCpyDest = 0;

			*pLineNext = 0L;
			/*0 -> there are NO more lines in the text buffer*/
			return 0;
		}else{
			/*copy line content into the supplied dest buffer
			check for buffer overflow*/

			if( (*charCount) < maxLen ){
				*ptrCpyDest = *ptrItemEnd;
				ptrCpyDest++;
				(*charCount)++;
			}else{

				DBGCRT("Line is longer then the max allowed size!\r\n");

				/*terminate dest buffer*/
				*ptrCpyDest = 0;

				*pLineNext = 0L;
				/*0 -> there are NO more lines in the text buffer! Error*/
				return 0;
			}

			ptrItemEnd++;
		}
	}/*while*/
}
```

### bgPVLogger2.c
```c
/********************************************************************
 * COPYRIGHT -- belgor
 ********************************************************************
 * Package: bglib
 * File: bgPVLogger.c
 * Author: goran
 * Created: October 13, 2011
 *******************************************************************/

#include <bur/plctypes.h>
#ifdef _DEFAULT_INCLUDES
#include <AsDefault.h>

/**
 Simple logging.
 Set to 0 when simple log is not needed
 To view this log, open Automation Studio  watch window and insert below defined
 logxx variable.
 Most recent log entry is always on the top (index 0)
 */
#if 1
//#include "bgsprintf.h"
//#include "bgsprintf.c"
#include "bgstring.h"
#include "bgstring.c"

typedef struct bgPVLogger_typ
{
	int initOk;
	char* logbuf;
	int entryCount;
	int entryLen;
}bgPVLogger_typ;

static void bgPVLoggerInit(bgPVLogger_typ* p, char* logbuf, int logEntryCount, int logEntryLen)
{
	if(!logbuf || !logEntryCount || !logEntryLen)
		return;

	p->logbuf = logbuf;
	p->entryCount = logEntryCount;
	p->entryLen = logEntryLen;
	p->initOk = 1;
}

static void shiftlog(bgPVLogger_typ* p)
{
int ii;
	if(!p || !p->initOk)
		return;

	for(ii=(p->entryCount-2); ii>=0; ii--){
		bgStrCpyN(&p->logbuf[(ii+1) * p->entryLen], &p->logbuf[ii * p->entryLen], p->entryLen);
	}
}

#define DBG(loggerInstance, format, args...)	shiftlog(&loggerInstance); snprintf2(&loggerInstance.logbuf[0], loggerInstance.entryLen, format, ## args);
//#define DBG(loggerInstance, format, args...)   ;
#define DBGINIT(loggerInstance,  logbuf, logEntryCount, logEntryLen) bgPVLoggerInit(&loggerInstance, &logbuf[0][0], logEntryCount, logEntryLen);

#else

#define DBG(loggerInstance, format, args...)   ;

#endif

#endif
```

### bgTcpSocketClient.c
```c
/*
File: bgTcpSocketClientServer.c
=====

B&R Libraries:
==============
Make sure to add following .a files to the task using this source file:
libsys_lib.a
libbrsystem.a
libastcp.a
*/

/*
B&R components:
===============================================================================
*/
#include <bur/plc.h>
#include <bur/plctypes.h>
#include <ethsock.h>
#include <astcp.h>
#include <brsystem.h>
#include <sys_lib.h>

/*
BG components
===============================================================================
*/
#include "bgdebug.h"
#include "bgstring.h"

#include "bgTcpSocketClientServer.h"
#include "bgHttpProtocol.h"

/*
Tcp Socket Client
*/
static void bgTcpSocketClientDefaultSessionHandler(bgTcpSocketSession_typ* pSession);
static void bgTcpSocketClientSessionStateMachine(bgTcpSocketSession_typ* pSession);
static void	bgTcpSocketClientExecuteSessionHandler(bgTcpSocketSession_typ* pSession, int init);

static void bgTcpSocketClientMemAlloc(bgTcpSocketClient_typ* pClient);
static void bgTcpSocketClientSessionStart(bgTcpSocketClient_typ* pClient);
static void	bgTcpSocketClientExecuteSessionHandler(bgTcpSocketSession_typ* pSession, int init);
static void bgTcpSocketClientSessionCyclic(bgTcpSocketClient_typ* pClient);
static void bgTcpSocketClientSessionLauncher(bgTcpSocketClient_typ* pClient);
static void setSocketAddressData(ETH_sockaddr_typ *adrData, char *hostIpAddressString, unsigned short hostPort);
static void swapBytesInShort(unsigned short *value);

/*
TCP Socket Client
######################################################################################################
######################################################################################################
######################################################################################################
######################################################################################################
*/
void bgTcpSocketClientInit(bgTcpSocketClient_typ* pClient,
    int sessionSendBufSize,
    int sessionRecvBufSize,
    int applicationBufSize,
    char* pRecvBuf,
    void (*pSessionHandler)(bgTcpSocketSession_typ*),
    void (*pApplicationHandler)(bgTcpSocketSession_typ*))
{
    pClient->serverPort = 0;

	pClient->recvBuffer = pRecvBuf;

	/*Recv buffer can't be allocated! recv DOES NOT WORK if the buffer is not in PV space!?!?!?!?*/
	if(!pRecvBuf){
		DBGCRT("bgTcpSocketClientInit: recvBuf not defined!\r\n");
		pClient->memAllocStatus2 = 1;
		return;
	}

    pClient->serverIpAddr[0] = 0;

    pClient->numSupportedSessions = 1;

    pClient->sessionSendBufSize = sessionSendBufSize;

    pClient->sessionRecvBufSize = sessionRecvBufSize;

	pClient->applicationBufSize = applicationBufSize;

	/*Recv buffer can't be allocated! recv DOES NOT WORK if the buffer is not in PV space!?!?!?!?*/
    pClient->sessionTotalBufSize = pClient->sessionSendBufSize + pClient->applicationBufSize;

    pClient->totalBufSize = pClient->sessionTotalBufSize * pClient->numSupportedSessions;

    pClient->pSessionHandler = pSessionHandler;

    pClient->pApplicationHandler = pApplicationHandler;

	pClient->sockStateData = BGTCPSOCK_STATE_NONE;

	pClient->dbgDumpSendBuf = 0;
	pClient->dbgDumpRecvBuf = 0;

	/*allocate memory for send/recv buffers*/
	bgTcpSocketClientMemAlloc(pClient);

	if(pClient->memAllocStatus2 ){
			DBGCRT("bgTcpSocketClientInit: memory error! memAllocStatus2=%d\r\n", pClient->memAllocStatus2);
	}
}

void bgTcpSocketClientCyclic(bgTcpSocketClient_typ* pClient)
{
int ret;
	/*non-blocking I/O control*/
static ETH_fd_set_typ fdR;
static ETH_fd_set_typ fdW;
static ETH_timeval_typ timeOut;

	/*if memalloc fails, can't do much!*/
	if(pClient->memAllocStatus2)
		return;

	/*monitor upper layer requests to start a client session*/
	bgTcpSocketClientSessionLauncher(pClient);

	/*execute session state machine*/
	bgTcpSocketClientSessionCyclic(pClient);

	/*client state machine*/
	switch(pClient->sockStateData){
		case BGTCPSOCK_STATE_NONE:
    		return;
		break;

		case BGTCPSOCK_STATE_INITOPEN:

 			/*create socket*/
			pClient->tcpOpen.ident = socket(ETH_AF_INET, ETH_SOCK_STREAM, 0);

			if( pClient->tcpOpen.ident == ERR_SOCKET ){
				DBGMSG("socket create error (init open); EthGetError=%d\r\n", EthGetError());
				pClient->sockStateData = BGTCPSOCK_STATE_NONE;
				break;
			}

			pClient->tcpClient.ident = pClient->tcpOpen.ident;
			pClient->tcpClose.ident = pClient->tcpOpen.ident;

			/*set non-blocking socket operation*/
			{
				UDINT arg = 1;
				ioctl(pClient->tcpOpen.ident, ETH_FIONBIO, (UDINT)&arg);
			}

#if 0
			/*get sock options*/
			{
				ret = getsockopt(pClient->tcpOpen.ident, ETH_SOL_SOCKET, ETH_SO_SNDTIMEO, (UDINT)&opt1, (UDINT)&opt1size);
				DBGMSG("getsockopt ret=%d\r\n", ret);
			}
#endif

			/*reset select flags*/
			fd_zero((UDINT)&fdR);
			fd_zero((UDINT)&fdW);

			/*set time-out to 10ms*/
			timeOut.tv_sec = 0;
			timeOut.tv_usec = 1000 * 10;

			pClient->sockStateData = BGTCPSOCK_STATE_OPEN;

		case BGTCPSOCK_STATE_OPEN:

			/*connect to remote host*/
			{
			ETH_sockaddr_typ serverAdr;
			setSocketAddressData(&serverAdr, pClient->serverIpAddr, pClient->serverPort);
			ret = connect(pClient->tcpOpen.ident, (UDINT)&serverAdr, sizeof(ETH_sockaddr_typ) );
			}

			if(ret == ERR_SOCKET){
				UINT errCode = EthGetError();
				if(errCode == ERR_ETH_INPROGRESS){
					/*next: wait connect to complete*/
					DBGMSG("socket connect - wait connect to complete!\r\n");
					pClient->sockStateData = BGTCPSOCK_STATE_CLIENT;
				    break;
				}else
				if(errCode == ERR_ETH_ISCONN){
					/*it's connected -> done*/
					DBGMSG("socket connect ok(1)!\r\n");
	                bgTcpSocketClientSessionStart(pClient);
					pClient->sockStateData = BGTCPSOCK_STATE_CONNECTED;
					break;
				}
				else{
					DBGMSG("socket connect error(open); EthGetError=%d\r\n", EthGetError());
					pClient->sockStateData = BGTCPSOCK_STATE_NONE;
					break;
				}
			}
			/*connected!*/
			/*it's connected -> done*/
			DBGMSG("socket connect ok(2)!\r\n");
            bgTcpSocketClientSessionStart(pClient);
			pClient->sockStateData = BGTCPSOCK_STATE_CONNECTED;
		break;
		case BGTCPSOCK_STATE_CLIENT:
			/*select waits for connection to complete*/
			fd_set(pClient->tcpOpen.ident, (UDINT)&fdR);
			fd_set(pClient->tcpOpen.ident, (UDINT)&fdW);
			ret = sock_select(32, (UDINT)&fdR, (UDINT)&fdW, 0L, (UDINT)&timeOut);

			if(ret == ERR_SOCKET){
				DBGMSG("socket connect error; (cli) EthGetError=%d\r\n", EthGetError());
				pClient->sockStateData = BGTCPSOCK_STATE_CLOSE;
				break;
			}

			if(ret == 0){

			}else{
				if( fd_isset(pClient->tcpOpen.ident, (UDINT)&fdW) ){
					DBGMSG("socket connect(long) ok!\r\n");
	                bgTcpSocketClientSessionStart(pClient);
					pClient->sockStateData = BGTCPSOCK_STATE_CONNECTED;
				}
			}
		break;
        case BGTCPSOCK_STATE_CONNECTED:
			/*Monitor session operation; generate OnResponseReady & OnResponseError triggers*/
            /*TODO: implement timeout here -> kill sessions if stuck*/
			if(pClient->session[0].socketState == BGTCPSOCK_SESSION_STATE_NONE){
				pClient->sockStateData = BGTCPSOCK_STATE_NONE;
			}
        break;
        case BGTCPSOCK_STATE_CLOSE:
			close(pClient->tcpClose.ident);
	    	pClient->sockStateData = BGTCPSOCK_STATE_NONE;
			DBGMSG("bgTcpSocketClientSessionStateMachine(): closing socket\r\n");
        break;
        case BGTCPSOCK_STATE_ERROR:
        break;
	 }

    return;
}

static void bgTcpSocketClientMemAlloc(bgTcpSocketClient_typ* pClient)
{
unsigned int memSize;
int i;

	/*Get System Memory Information*/
	pClient->MEMInfo.enable = 1;
	MEMInfo(&pClient->MEMInfo);

	memSize = pClient->totalBufSize;

	/*allocate space for send/recv buffers*/
	if(pClient->sendRecvBuffer == 0){
		/* allocate new memory from RAM*/
    	pClient->memAllocStatus2 = TMP_alloc(memSize, (void**)&pClient->sendRecvBuffer);
	}else{
		/*memory is allready allocated -> free it first!*/
    	pClient->memAllocStatus2 = TMP_free(memSize, (void**)pClient->sendRecvBuffer);

    	/*allocate new memory from RAM*/
    	pClient->memAllocStatus2 = TMP_alloc(memSize, (void**)pClient->sendRecvBuffer);
	}

	/*assign send/recv buffer ptrs*/
    pClient->session[0].pSendBuf = (char*)(pClient->sendRecvBuffer + i * pClient->sessionTotalBufSize);
	pClient->session[0].sendBufLength = pClient->sessionSendBufSize;

    pClient->session[0].pAppBuf = (char*)(pClient->session[0].pSendBuf + pClient->sessionSendBufSize);
	pClient->session[0].appBufLength = pClient->applicationBufSize;

    pClient->session[0].pRecvBuf = pClient->recvBuffer;
	pClient->session[0].recvBufLength = pClient->sessionRecvBufSize;
}

static void bgTcpSocketClientSessionStart(bgTcpSocketClient_typ* pClient)
{
int i;
bgTcpSocketSession_typ *pSession;

	/* client: pClient->numSupportedSessions = 1 ALWAYS!*/
    for(i=0; i < pClient->numSupportedSessions; i++){
        if( pClient->session[i].socketState == BGTCPSOCK_SESSION_STATE_NONE){
            pSession = &pClient->session[i];
            pSession->socketState = BGTCPSOCK_SESSION_STATE_SEND;

			pSession->tcpSend.enable = 1;
			pSession->tcpSend.ident = pClient->tcpOpen.ident;   		/* copy the  Ident number */
			pSession->tcpSend.flags = 0;
			pSession->tcpSend.pData = (UDINT)pSession->pSendBuf;

			pSession->tcpRecv.enable = 1;
			pSession->tcpRecv.ident = pClient->tcpOpen.ident;     		/* copy the  Ident number */

			pSession->tcpRecv.pData = (UDINT)pSession->pRecvBuf;        /* address of the buffer */;

			pSession->tcpRecv.datamax = pClient->sessionRecvBufSize;    /* length of the buffer */;

			pSession->tcpClose.enable = 1;
   			pSession->tcpClose.ident = pClient->tcpOpen.ident;    		/* copy the  Ident number */

			pSession->pTcpLayer = (char*)pClient;	                    /*session has ptr to tcp layer*/

            pSession->rxByteCount = 0;
            strcpy(pSession->clientIpAddr, pClient->clientIpAddr);

			pSession->dbgDumpRecvBuf = pClient->dbgDumpRecvBuf;
			pSession->dbgDumpSendBuf = pClient->dbgDumpSendBuf;

			/*init session specific handler - call the handler with init pSession->flag=1*/
			bgTcpSocketClientExecuteSessionHandler(pSession, 1);

			DBGMSG("bgTcpSocketClientSessionStart(): connection to %s, starting session Id= %d\r\n", pClient->serverIpAddr, i);
            return;
        }
    }

	DBGCRT("bgTcpSocketClientSessionStart(): client busy! activeSessions= %d\r\n", pClient->numSupportedSessions);
    pClient->sockStateData = BGTCPSOCK_STATE_TOOBUSY;
}

static void	bgTcpSocketClientExecuteSessionHandler(bgTcpSocketSession_typ* pSession, int init)
{
bgTcpSocketClient_typ* pClient = (bgTcpSocketClient_typ*)pSession->pTcpLayer;

	pSession->init = 0;
	if( init )
		pSession->init = 1;

	DBGMSG("bgTcpSocketClientExecuteSessionHandler\r\n p1=%d p2=%d\r\n", pClient->pSessionHandler, bgHttpClientSessionHandler);

/*
	bgHttpClientSessionHandler(pSession);
*/
    if(pClient->pSessionHandler)
    	(*pClient->pSessionHandler)(pSession);
    else
    	bgTcpSocketClientDefaultSessionHandler(pSession);

	pSession->init = 0;
}

static void bgTcpSocketClientSessionCyclic(bgTcpSocketClient_typ* pClient)
{
int i;
bgTcpSocketSession_typ *pSession;
int activeSessions = 0;

    for(i=0; i < pClient->numSupportedSessions; i++){
        pSession = &pClient->session[i];

        if( pSession->socketState != BGTCPSOCK_SESSION_STATE_NONE){
            activeSessions++;
            bgTcpSocketClientSessionStateMachine(pSession);
        }
    }
    pClient->numActiveSessions = activeSessions;
}

static void bgTcpSocketClientSessionLauncher(bgTcpSocketClient_typ* pClient)
{
int i;
bgTcpSocketSession_typ *pSession;

    for(i=0; i < pClient->numSupportedSessions; i++){
        pSession = &pClient->session[i];

		if( (pSession->bSendData) ){
			pSession->bSendData = 0;
			if(pClient->sockStateData == BGTCPSOCK_STATE_NONE){
				pClient->sockStateData = BGTCPSOCK_STATE_INITOPEN;
			}else{
				DBGMSG("bgTcpSocketClientSessionLauncher: client session start rejected; client is busy! cliState=%d\r\n",
					pClient->sockStateData);
			}
		}
    }
}
static void bgTcpSocketClientSessionStateMachine(bgTcpSocketSession_typ* pSession)
{
int ret;

    switch(pSession->socketState){
		case BGTCPSOCK_SESSION_STATE_SEND:

        	ret = send(pSession->tcpSend.ident, (UDINT)pSession->pSendBuf, pSession->tcpSend.datalen, 0L);

        	if(ret == ERR_SOCKET){
				DBGMSG("send error EthGetError=%d\r\n", EthGetError());
				pSession->socketState = BGTCPSOCK_SESSION_STATE_CLOSE;    /*close this socket*/
				return;
        	}

			/*remember the send length*/
			DBG("send() ok; bytes=%d\r\n", (int)ret);
			pSession->tcpSend.sentlen = ret;
	   		pSession->socketState = BGTCPSOCK_SESSION_STATE_RECEIVE;    /*close this socket session*/

		/*break;*/

		case BGTCPSOCK_SESSION_STATE_RECEIVE:
	       	/*call receive (NON BLOCKING MODE!)*/
        	ret = recv(pSession->tcpRecv.ident, (UDINT)pSession->tcpRecv.pData, pSession->tcpRecv.datamax, 0L);

        	if(ret == ERR_SOCKET){
        		UINT errCode = EthGetError();
        		/*none blocking receive return this following value if data is not available yet*/
        		if( errCode == ERR_ETH_WOULDBLOCK ){
        			/*wait response*/
					return;
        		}
				DBGMSG("RxError EthGetError=%d\r\n", errCode);
	   			pSession->socketState = BGTCPSOCK_SESSION_STATE_CLOSE;    /*close this socket session*/
				break;
        	}

			pSession->tcpRecv.recvlen = ret;

            if(pSession->tcpRecv.recvlen){
				DBGMSG("rx OK! rxLen=%d\r\n", ret);

				bgTcpSocketClientExecuteSessionHandler(pSession, 0);

				/*uper layer completed processing? */
				if( pSession->bCloseSession){
					pSession->bCloseSession = 0;
	   					pSession->socketState = BGTCPSOCK_SESSION_STATE_CLOSE;    /*close this socket session*/
				}
            }else{
				DBGMSG("bgTcpSocketClient..: RMT SOCK CLOSED!\r\n");
	   			pSession->socketState = BGTCPSOCK_SESSION_STATE_CLOSE;    /*close this socket session*/
			}
			return;
		break;

		case BGTCPSOCK_SESSION_STATE_CLOSE:
			close(pSession->tcpClose.ident);
	    	pSession->socketState = BGTCPSOCK_SESSION_STATE_NONE;
			DBGMSG("bgTcpSocketClientSessionStateMachine(): stopping session Id= %d\r\n", pSession->ident);
		break;

		case BGTCPSOCK_SESSION_STATE_DELAY:
			pSession->delayCounter--;
			if(pSession->delayCounter <= 0)
    			pSession->socketState = BGTCPSOCK_SESSION_STATE_CLOSE;    /*close this server socket*/
		break;

		default:

		break;
	}
}

#if 0
static void bgTcpSocketClientSessionSendData(bgTcpSocketSession_typ* pSession, int len)
{
	pSession->tcpSend.datalen = len;
	pSession->socketState = BGTCPSOCK_STATE_INITOPEN;

#if 0
{
int i;
char text[90];
/*session/application/protocol specific data structure*/
httpRequest_typ* r = (httpRequest_typ*)pSession->pProtocol;

	DBGMSG("bgHttpSend(): lenght(bytes): total=%d(%d) header=%d content=%d\r\n",
		len, r->sendTotalLength, r->sendHeaderLength, r->sendContentLength);

	DBGMSG("bgHttpSend dump:\r\n");
	DBGMSG("============================================\r\n");
	for(i=0;i<len; i++){
 		if( ((i+1)*80) < len ){
			memcpy(&text[0], &pSession->pSendBuf[i*80], 80);
			text[80]=0;
			DBGMSG("%s", &text[0]);
		}else{
			memcpy(&text[0], &pSession->pSendBuf[i*80], len - (i*80));
			text[len - (i*80)]=0;
			DBGMSG("%s", &text[0]);
			break;
		}
	}
	DBGMSG("============================================\r\n\r\n");
}
#endif

}
#endif
/*
Default session handler
######################################################################################################
######################################################################################################
######################################################################################################
######################################################################################################
*/
static void bgTcpSocketClientDefaultSessionHandler(bgTcpSocketSession_typ* pSession)
{
    /*default session handler -> send out http error response "internal server error"*/
/*    httpSendErrorResponse(pSession, 500);
*/
}

static void setSocketAddressData(ETH_sockaddr_typ *adrData, char *hostIpAddressString, unsigned short hostPort)
{

	unsigned short sin_family;
	unsigned short family;
	unsigned short length;
	unsigned short port;

	family = ETH_AF_INET;
	length = sizeof(ETH_sockaddr_typ);
	sin_family = (family << 8) + length;

	adrData->sin_family = sin_family;
	port = hostPort;
	swapBytesInShort(&port);
	adrData->sin_port = port;
	if( strlen(hostIpAddressString) < 8)
		adrData->sin_addr = ETH_INADDR_ANY;
	else
		adrData->sin_addr = inet_addr( (unsigned long) hostIpAddressString);
	adrData->sin_zero[0]=0;
	adrData->sin_zero[1]=0;
	adrData->sin_zero[2]=0;
	adrData->sin_zero[3]=0;
	adrData->sin_zero[4]=0;
	adrData->sin_zero[5]=0;
	adrData->sin_zero[6]=0;
	adrData->sin_zero[7]=0;
}

static void swapBytesInShort(unsigned short *value)
{

union{
	unsigned short 	shortValue;
	unsigned char	bytes[2];
}swapValue;

unsigned char tempByte;

	swapValue.shortValue = *value;
	tempByte = swapValue.bytes[0];
	swapValue.bytes[0] = swapValue.bytes[1];
	swapValue.bytes[1] = tempByte;
	*value = swapValue.shortValue;
}
```

### HMIalert.typ - Global data types
```iecst
(********************************************************************
 * COPYRIGHT -- piedmont
 ********************************************************************
 * Package: HMI
 * File: HMI.typ
 * Author: goran
 * Created: August 28, 2013
 ********************************************************************
 * Data types of package HMI
 ********************************************************************)
(*########################################################################*)
(*HMI object - ALERT*)
(*########################################################################*)

TYPE
	hmiAlert_typ : 	STRUCT
		message : STRING[512];
		color_idx : USINT;
		header : STRING[128];
		type : UINT; (*0-info; 1-warning; 2-error*)
		status : UINT; (*Status for common dialog layer*)
		tmr1RemainingTimeSec : UDINT; (*Timer remaining time (sec)*)
		tmr1 : TON; (*Dialog control timer*)
	END_STRUCT;
END_TYPE
```

### HMI.typ - Global data types
```iecst
(********************************************************************
 * COPYRIGHT -- piedmont
 ********************************************************************
 * Package: HMI
 * File: HMI.typ
 * Author: goran
 * Created: August 28, 2013
 ********************************************************************
 * Data types of package HMI
 ********************************************************************)
(*########################################################################*)
(*HMI key assinged PV-s (i.e. page navigation, save btns, etc)*)
(*########################################################################*)

TYPE
	hmiControlLogicKeys_typ : 	STRUCT
		btnRestartLoginTimer : USINT; (*1-means that login timer restart is requested*)
		btnLoginIcon : USINT; (*1-means that login logo (icon) is pressed*)
		menuKeyPressLT : ARRAY[0..HMI_ENUM_MENU_ITEMS_LT]OF BOOL; (*Mom keys connected to menu items LF*)
		menuKeyPressRT : ARRAY[0..HMI_ENUM_MENU_ITEMS_RT]OF BOOL; (*Mom keys connected to menu items RT*)
	END_STRUCT;
END_TYPE

(*########################################################################*)
(*HMI navigation PV-s (i.e. PV-s assigned to required VC PV-s such as currentPage, etc)*)
(*########################################################################*)

TYPE
	hmiNavigationLogic_typ : 	STRUCT
		changePage : USINT;
		currentPage : USINT;
		htmlCurrentURL : STRING[127];
		htmlChangeURL : STRING[127];
		currentPageText : STRING[31];
		prevPage : USINT;
		nextPage : USINT;
		pageInit : BOOL;
		pageExit : BOOL;
		state : USINT;
		currentStateText : STRING[31];
		statePrev : USINT;
		stateNext : USINT;
		loginLevel : UDINT;
		stateInit : BOOL;
		tmr1 : TON; (*Alert message control timer*)
		tmr2 : TON; (*Unack alarms message alert blinking timer*)
		tmr3 : TON; (*Password level reset timer*)
		tmr3RemainingTimeSec : UDINT;
		tmr3RemainingTimeMin : UDINT;
		tmr4 : TON;
	END_STRUCT;
END_TYPE

(*########################################################################*)
(*HMI related status control PV-s (i.e. visibility, locking, etc)*)
(*########################################################################*)

TYPE
	hmiControlLogicStatus_typ : 	STRUCT
		visibleSaveCfg : UINT;
		menuVisibleLT : UINT; (*Main menu LF visibility control *)
		menuVisibleRT : UINT; (*Main menu RT visibility control *)
		menuVisibleRTItems : ARRAY[0..HMI_ENUM_MENU_ITEMS_RT]OF UINT; (*Main menu items RT visibility control - for buttons stacked on top of each other in the upper, rt *)
		menuIndexLT : UINT; (*Main menu currently selected menu item - LF*)
		show_motion_tab : USINT;
		show_Aux_tab : USINT;
		show_io_tab : UINT;
		menuIndexRT : UINT; (*Main menu currently selected menu item - RT*)
		loginVisibleGE1 : USINT; (*Visibility control for login level related stuff - set to visible (0) if login level >= 1; othervise set to 1 (i.e. loginLevel < 1)*)
		loginVisibleGE2 : USINT; (*Visibility control for login level related stuff - set to visible (0) if login level >= 2; othervise set to 1 (i.e. loginLevel < 2)*)
		loginVisibleGE3 : USINT; (*Visibility control for login level related stuff - set to visible (0) if login level >= 2; othervise set to 1 (i.e. loginLevel < 2)*)
		menuLFHideTimer : TON; (*timer of automaticaly hiding LF dropdown menu*)
		menuRTHideTimer : TON; (*timer of automaticaly hiding RT dropdown menu*)
		tabKeysRadioDataPoint : USINT; (*DP that tab button are writing to in order to create radio buttons/tab view effect*)
		tabKeysRadioArray : ARRAY[0..HMI_ENUM_TAB_KEYS_MAX]OF USINT;
		tabKeysToggle : ARRAY[0..HMI_ENUM_MENU_ITEMS_LT]OF USINT;
		passwordStrings : ARRAY[0..HMI_PWD_LEVELS]OF STRING[HMI_PWD_MAXLEN]; (*Password strings used for loginLevel control*)
	END_STRUCT;
END_TYPE

(*=============================================================================*)
(*Recipe related HMI logic.*)
(*=============================================================================*)

TYPE
	hmiRecipeLogic_typ : 	STRUCT
		recVisible : USINT; (*Recipe related visibility control*)
		recSelectIdx : UINT; (*Recipe list index*)
		recSelectIdxMax : UINT; (*Recipe list index*)
		recSaveAsIdx : UINT; (*Recipe index for SaveAs action*)
		recSelectName : STRING[80]; (*Name of the currently selected recipe from the recipe list*)
		btnLockedActivate : USINT; (*Button lock control*)
		btnLockedNew : USINT; (*Button lock control*)
		btnLockedDelete : USINT; (*Button lock control*)
		btnLockedSaveAs : USINT; (*Button lock control*)
		btnActivate : BOOL; (*mom btn to Activate a recipe*)
		btnNew : BOOL; (*mom btn to New a recipe*)
		btnDelete : BOOL; (*mom btn to Delete a recipe*)
		btnSaveAs : BOOL; (*mom btn to SaveAs a recipe*)
		stateRecipes : UDINT;
	END_STRUCT;
END_TYPE

(*=============================================================================*)
(*Fileio Items*)
(*=============================================================================*)
(*=============================================================================*)
(*Tabs Control*)
(*=============================================================================*)
(*=============================================================================*)
(*HMI related navigation and control logic.*)
(*=============================================================================*)
(*Insert your comment here.*)
(*Insert your comment here.*)

TYPE
	hmiTableRecCfgTrigger_typ : 	STRUCT
		Control : BOOL;
		Dispense : BOOL;
	END_STRUCT;
	hmiTableTrigger_typ : 	STRUCT
		Rec : hmiTableRecCfgTrigger_typ;
		Cfg : hmiTableRecCfgTrigger_typ;
	END_STRUCT;
	hmiTableLoad_typ : 	STRUCT
		Trigger : BOOL;
	END_STRUCT;
	hmiTables_typ : 	STRUCT
		Trigger : hmiTableTrigger_typ;
		Load : hmiTableLoad_typ;
	END_STRUCT;
END_TYPE

(*Insert your comment here.*)

TYPE
	hmiControlLogic_typ : 	STRUCT
		status : hmiControlLogicStatus_typ;
		keys : hmiControlLogicKeys_typ;
		prv : hmiNavigationLogic_typ; (*Hmi (panel) private data for handling screen navigation and hmi logic. Used only wihin HMI.*)
		recipes : hmiRecipeLogic_typ;
		alertMsg : hmiAlert_typ;
		dialogMsg : hmiDialog_typ;
		tables : hmiTables_typ;
	END_STRUCT;
END_TYPE
```

### HMI.var - Global variables
```iecst
(********************************************************************
 * COPYRIGHT -- piedmont
 ********************************************************************
 * Package: HMI
 * File: HMI.var
 * Author: goran
 * Created: August 28, 2013
 ********************************************************************
 * Variables of package HMI
 ********************************************************************)
VAR CONSTANT
	HMI_ENUM_FORCEIO_LASTINDEX : USINT := 7;
END_VAR
VAR
	gHmiParamTable : hmiParamListTable_typ := (0); (*Machine configuration / parameter settings logic *)
	gHmi : hmiControlLogic_typ := (0); (*HMI logic, page navigation, visibility control, etc.*)
	gHmiMsgScroll : hmiMsgScrolling_typ := (0); (*Scrolling Alarm Msg Support*)
	gHMIForceIO : hmiForceIO_typ := (0);
END_VAR
```

### Program Logical/HMI/hmilogic (ANSIC) - Service that manages navigating through the VC4 HMI

#### hmiAlert.h
```c
/********************************************************************
 * COPYRIGHT -- piedmont
 ********************************************************************
 * Program: hmilogic
 * File: hmiAlert.h
 * Author: goran
 * Created: September 05, 2013
 *******************************************************************/

#include <bur/plctypes.h>
#ifdef _DEFAULT_INCLUDES
#include <AsDefault.h>
#endif
void hmiAlertHide(hmiAlert_typ* p);
BOOL hmiAlertIsActive(hmiAlert_typ* p);
void hmiAlertShow(hmiAlert_typ* p, char* alertText, UDINT alertDuration);
void hmiAlertCyclic(hmiAlert_typ* p);
```

#### hmiParamList.h
```c
/********************************************************************
 * COPYRIGHT -- piedmont
 ********************************************************************
 * Program: hmilogic
 * File: hmiParamList.h
 * Author: goran
 * Created: September 05, 2013
 *******************************************************************/
#include <bur/plctypes.h>
#ifdef _DEFAULT_INCLUDES
#include <AsDefault.h>
#endif
//void hmiParamListTableCyclic(hmiParamListTable_typ* p);
void hmiParamListTableEntryLast(hmiParamListTable_typ* p);
void hmiParamListTableEntryFirst(hmiParamListTable_typ* p, char* pListName);
 void hmiParamListTableAddEntryNext(hmiParamListTable_typ* p, UDINT pValue, char* pName, REAL valDefault, REAL valMin, REAL valMax, int decPlaces, REAL k_factor, REAL n_factor, UINT valueType, char* pDescription);
```

#### loginLogic_Header.h
```c
#include <bur/plctypes.h>
#ifdef _DEFAULT_INCLUDES
#include <AsDefault.h>
#endif

void	loginLevelLogicCyclic();
void loginLevelParameterEditControl(UDINT minLevel);
```

### Program Logical/HMI/ForceIO (IEC)

#### Main.st
```iecst
PROGRAM _INIT

	gHMIForceIO.forceItems[0].pAddrIO := ADR(IO.oCreaserCCWRotation);
	gHMIForceIO.forceItems[1].pAddrIO := ADR(IO.oCreaserCWRotation);
	gHMIForceIO.forceItems[2].pAddrIO := ADR(IO.oBoardFeedingLight);
	gHMIForceIO.forceItems[3].pAddrIO := ADR(IO.oUIIndicatorLight);

	gHMIForceIO.forceItems[4].pAddrIO := ADR(IO.iSafeMachineState);
	gHMIForceIO.forceItems[5].pAddrIO := ADR(IO.iCreaserShaftSensor);
	gHMIForceIO.forceItems[6].pAddrIO := ADR(IO.iFiberOpticSensor);
	gHMIForceIO.forceItems[7].pAddrIO := ADR(IO.iSM1Disabled);
END_PROGRAM

PROGRAM _CYCLIC
	IF gHMIForceIO.forceEnable = 0 THEN
		gHMIForceIO.forceItemsVisibility := 1;

		FOR ii_force := 0 TO HMI_ENUM_FORCEIO_LASTINDEX BY 1 DO
			pForceIOPt ACCESS gHMIForceIO.forceItems[ii_force].pAddrIO;
			pSet ACCESS ADR(gHMIForceIO.forceItems[ii_force].set);
			pReset ACCESS ADR(gHMIForceIO.forceItems[ii_force].reset);
			pToggle ACCESS ADR(gHMIForceIO.forceItems[ii_force].toggle);

			pSet := FALSE;
			pReset := FALSE;
			pToggle := FALSE;
		END_FOR;
	ELSE
		gHMIForceIO.forceItemsVisibility := 0;

		FOR ii_force := 0 TO HMI_ENUM_FORCEIO_LASTINDEX BY 1 DO
			IF gHMIForceIO.forceItems[ii_force].pAddrIO <> 0 THEN
				pForceIOPt ACCESS gHMIForceIO.forceItems[ii_force].pAddrIO;
				pSet ACCESS ADR(gHMIForceIO.forceItems[ii_force].set);
				pReset ACCESS ADR(gHMIForceIO.forceItems[ii_force].reset);
				pToggle ACCESS ADR(gHMIForceIO.forceItems[ii_force].toggle);

				IF pSet THEN
					pForceIOPt := TRUE;
				END_IF;

				IF pReset THEN
					pForceIOPt := FALSE;
				END_IF;

				IF pToggle THEN
					pToggle := FALSE;
					pForceIOPt := NOT pForceIOPt;
				END_IF;
			END_IF;
		END_FOR;
	END_IF;

END_PROGRAM

PROGRAM _EXIT
	(* Insert code here *)

END_PROGRAM
```

### Program Logical/HMI/HMITableManager (IEC) - Manage activating the PV List tables for recipe, configuration params (gRecCfg.active.<>)

#### Variables.var
```iecst
VAR
	Init_Logbook : FBK_Init_Logbook;
	loadHMITable : ARRAY[0..DEFINE_MAX_IDX_HMI_TABLES] OF hmiTableFBK_typ;
	tableStats : hmiTableStats_typ;
END_VAR
```

- Visualisation Logical/HMI/Visu (not shown)

### Program Logical/HMI/HMI_Alarms

#### Cyclic.st
```iecst
PROGRAM _CYCLIC
	brsmemcpy(ADR(AppAlarms.AlarmImage[0]), 	ADR(gAlarms), 					SIZEOF(Machine_Alarms_typ));

	brsmemcpy(ADR(gAcknowledge), 				ADR(AppAlarms.AlarmImage[0]), 	SIZEOF(Machine_Alarms_typ));

//	tmp_alarm_counter := 0;
//
//	FOR ii_alarms := 0 TO MAX_IDX_ALARMS BY 1 DO
//		IF gMachine.HMI.AlarmControls.Dispense.AlarmImage[ii_alarms] THEN
//			tmp_alarm_counter := tmp_alarm_counter + 1;
//		END_IF;
//
//		IF gMachine.HMI.AlarmControls.Inspect.AlarmImage[ii_alarms] THEN
//			tmp_alarm_counter := tmp_alarm_counter + 1;
//		END_IF;
//
//		IF gMachine.HMI.AlarmControls.Sensor.AlarmImage[ii_alarms] THEN
//			tmp_alarm_counter := tmp_alarm_counter + 1;
//		END_IF;
//
//		IF gMachine.HMI.AlarmControls.Safety.AlarmImage[ii_alarms] THEN
//			tmp_alarm_counter := tmp_alarm_counter + 1;
//		END_IF;
//
//		IF gMachine.HMI.AlarmControls.RecCfg.AlarmImage[ii_alarms] THEN
//			tmp_alarm_counter := tmp_alarm_counter + 1;
//		END_IF;
//
//		IF gMachine.HMI.AlarmControls.Hardware.AlarmImage[ii_alarms] THEN
//			tmp_alarm_counter := tmp_alarm_counter + 1;
//		END_IF;
//
//		IF gMachine.HMI.AlarmControls.Motor.AlarmImage[ii_alarms] THEN
//			tmp_alarm_counter := tmp_alarm_counter + 1;
//		END_IF;
//	END_FOR;

//	IF gAlarmResetRequested THEN
//		brsmemset(ADR(gAlarms.Dispense), 								0, 		SIZEOF(HERNON_Alarm_Dispense_typ));
//		brsmemset(ADR(gAlarms.Inspect), 								0, 		SIZEOF(HERNON_Alarm_Inspect_typ));
//		brsmemset(ADR(gAlarms.Sensor), 									0, 		SIZEOF(HERNON_Alarm_Sensor_typ));
//		brsmemset(ADR(gAlarms.Safety), 									0, 		SIZEOF(HERNON_Alarm_Safety_typ));
//		brsmemset(ADR(gAlarms.RecCfg), 									0, 		SIZEOF(HERNON_Alarm_RecCfg_typ));
//		brsmemset(ADR(gAlarms.Hardware), 								0, 		SIZEOF(HERNON_Alarm_HW_typ));
//		brsmemset(ADR(gAlarms.Motor), 									0, 		SIZEOF(HERNON_Alarm_Motor_typ));
//		gMachine.App.MotorVar.ChainDrive.Current.oError := FALSE;
//		gAlarmResetRequested := FALSE;
//	END_IF;
//
//	IF Alarm_Control.ActiveAlarms = 0 AND Alarm_Control.PendingAlarms = 0 AND tmp_alarm_counter = 0 THEN
//		gAlarmState := 0;
//	ELSIF Alarm_Control.ActiveAlarms = 0 AND Alarm_Control.PendingAlarms = 0 AND tmp_alarm_counter > 0 THEN
//		gAlarmState := 1;
//	ELSIF Alarm_Control.ActiveAlarms = 0 AND Alarm_Control.PendingAlarms > 0 THEN
//		gAlarmState := 2;
//	ELSE
//		gAlarmState := 3;
//	END_IF;

	AppAlarms_FBK();
//
//	gMachine.HMI.Dashboard.Application_Errors_Active := tmp_alarm_counter;
//	gMachine.HMI.Dashboard.System_Alarms_Active := Alarm_Control.ActiveAlarms;
//	gMachine.HMI.Dashboard.System_Alarms_Pending := Alarm_Control.PendingAlarms;
END_PROGRAM
```

- Project.language (not shown)

### Package Logical/Axisobj - Axisobj

### Axisi.ax
```
InitParameter (Version=3.16.1, NcSwId=ACP10)
  ACP10AXIS_typ:
    dig_in:
      level:
        reference = ncACTIV_HI
        pos_hw_end = ncACTIV_HI
        neg_hw_end = ncACTIV_HI
        trigger1 = ncACTIV_HI
        trigger2 = ncACTIV_HI
    encoder_if:
      parameter:
        count_dir = ncSTANDARD
        scaling:
          load:
            units = 1000
            rev_motor = 1
    limit:
      parameter:
        v_pos = 10000.0
        v_neg = 10000.0
        a1_pos = 50000.0
        a2_pos = 50000.0
        a1_neg = 50000.0
        a2_neg = 50000.0
        t_jolt = 0.0
        t_in_pos = 0.0
        pos_sw_end = 2000000000
        neg_sw_end = -2000000000
        ds_warning = 500.0
        ds_stop = 1000.0
        a_stop = 1.0E+30
        dv_stop = 0.0
        dv_stop_mode = ncOFF
    controller:
      mode = ncPOSITION
      position:
        kv = 50.0
        tn = 0.0
        t_predict = 0.0004
        t_total = 0.0004
        p_max = 1.0E+30
        i_max = 0.0
      speed:
        kv = 2.05
        tn = 0.0
        t_filter = 0.0
        isq_filter1:
          type = ncOFF
          a0 = 0.0
          a1 = 0.0
          b0 = 0.0
          b1 = 0.0
          b2 = 0.0
          c0_par_id = 0
          c1_par_id = 0
        isq_filter2:
          type = ncOFF
          a0 = 0.0
          a1 = 0.0
          b0 = 0.0
          b1 = 0.0
          b2 = 0.0
          c0_par_id = 0
          c1_par_id = 0
        isq_filter3:
          type = ncOFF
          a0 = 0.0
          a1 = 0.0
          b0 = 0.0
          b1 = 0.0
          b2 = 0.0
          c0_par_id = 0
          c1_par_id = 0
      uf:
        type = ncLINEAR
        auto_config = ncMOTOR_PAR
        u0 = 0.0
        un = 0.0
        fn = 50.0
        k_f_slip = 0.0
      ff:
        torque_load = 0.0
        torque_pos = 0.0
        torque_neg = 0.0
        kv_torque = 0.0
        inertia = 0.0
        t_filter_a = 0.0
    move:
      stop:
        parameter[0]:
          decel_ramp = ncA_LIMIT
          controller = ncON
        parameter[1]:
          decel_ramp = ncA_LIMIT
          controller = ncON
        parameter[2]:
          decel_ramp = ncA_LIMIT
          controller = ncON
        parameter[3]:
          decel_ramp = ncA_LIMIT
          controller = ncON
        quickstop:
          decel_ramp = ncA_LIMIT
        drive_error:
          decel_ramp = ncA_LIMIT
      homing:
        parameter:
          s = 0
          v_switch = 5000.0
          v_trigger = 500.0
          a = 50000.0
          mode = ncDIRECT
          edge_sw = ncPOSITIVE
          start_dir = ncPOSITIVE
          trigg_dir = ncPOSITIVE
          ref_pulse = ncOFF
          fix_dir = ncOFF
          tr_s_block = 0.0
          torque_lim = 0.0
          ds_block = 0.0
          ds_stop = 0.0
      basis:
        parameter:
          v_pos = 5000.0
          v_neg = 5000.0
          a1_pos = 50000.0
          a2_pos = 50000.0
          a1_neg = 50000.0
          a2_neg = 50000.0
    message:
      text:
        parameter:
          format = ncBREAK + ncZERO
          columns = 80
          data_modul = acp10etxen
```

### IO_Structures.typ - not listed in the package file held
```iecst
TYPE
	AS3500_Cure_IO_typ : 	STRUCT
		oUVCureChannel : ARRAY[0..1]OF BOOL;
		iUVCuringChannelOK : ARRAY[0..1]OF BOOL;
	END_STRUCT;
	StatusColors_typ : 	STRUCT
		Red : BOOL;
		Green : BOOL;
		Blue : BOOL;
	END_STRUCT;
	ErrorIO_typ : 	STRUCT
		oQuitError : BOOL;
		iErrorStatus : BOOL;
	END_STRUCT;
	AS5300_Encoder_Status_typ : 	STRUCT
		CycleTimeViolation : ErrorIO_typ;
		DataError : ErrorIO_typ;
		BWChannel : ErrorIO_typ;
		iPowerSupply : ARRAY[0..1]OF BOOL;
	END_STRUCT;
	AS5300_Dispense_Status_typ : 	STRUCT
		EdgeDetect : ErrorIO_typ;
	END_STRUCT;
	AS3500_Status_IO_typ : 	STRUCT
		iProcessStopRelay : ARRAY[0..1]OF BOOL;
		oStatusColor : StatusColors_typ;
		oSystemNeedsAttention : BOOL;
		oRunningReady : BOOL;
		iClearError : BOOL;
		Encoder : AS5300_Encoder_Status_typ;
		Dispense : AS5300_Dispense_Status_typ;
	END_STRUCT;
	AS5300_Inspection_typ : 	STRUCT
		oInspectionValid : BOOL;
		oInspectionGood : BOOL;
	END_STRUCT;
	AS3500_Control_IO_typ : 	STRUCT
		oTargetPresent : BOOL;
		iRunCmd : BOOL;
		iEncoderValue : UINT;
		iReservoirLevel : BOOL;
		iTargetPiP : BOOL;
		Inspection : AS5300_Inspection_typ;
		iX2XNettime : DINT;
		PiP_Sensor_Debounce : Debounce_Signal;
	END_STRUCT;
END_TYPE
```

### MachineControl.typ - not listed in the package file held
```iecst
TYPE
	AS3500HS_SM_States_Enum :
		(
		STATE_INIT := 0,
		STATE_IDLE := 1,
		STATE_RUNNING := 2,
		STATE_ERROR := 3
		);
	AS3500HS_ColorBar_Enum :
		(
		COLOR_NONE := 0,
		COLOR_GREEN_FLASH := 1,
		COLOR_GREEN := 2,
		COLOR_GREEN_BLUE_ALTERNATE := 3,
		COLOR_RED := 4,
		COLOR_GREEN_RED_ALTERNATE := 5
		);
END_TYPE

(*Insert your comment here.*)

TYPE
	Dispense_Control_Var_typ : 	STRUCT
		Current_Target_At_Dispense_Unit : UDINT;
		Target_Fractional_Position_Pct : REAL;
	END_STRUCT;
	AS3500HS_Control_Var_typ : 	STRUCT
		Dispense : ARRAY[0..MAX_IDX_VALVES]OF Dispense_Control_Var_typ;
	END_STRUCT;
	AS3500HS_Control_Alarms_typ : 	STRUCT
		Invalid_Par : USINT;
		Valve_Not_Ready : USINT;
		Encoder_Sim_Active : USINT;
	END_STRUCT;
	HERNON_Alarms_typ : 	STRUCT
		Control : AS3500HS_Control_Alarms_typ;
		Sureshot3500 : ARRAY[0..MAX_IDX_VALVES]OF HERNON_Alarm_Dispense_typ;
	END_STRUCT;
	AS3500HS_Position_Var_typ : 	STRUCT
		Home_Position : UINT;
		Ticks_Per_Target : UINT;
		Single_Turn_Rel_Home : UINT;
		Single_Turn_Absolute : UINT;
		Current_Target : UINT;
		Ticks_Within_Current_Target : UINT;
		Degrees_Absolute : REAL;
		Degrees_Rel_Home : REAL;
		Home_Position_Degrees : REAL;
		Target_Fractional_Position_Pct : REAL;
	END_STRUCT;
	AS3500HS_Dial_Vel_Calc : 	STRUCT
		Encoder_Counts_Per_Second : REAL;
		Deg_Per_S : REAL;
		RPM : REAL;
		Rev_Per_S : REAL;
		Targ_Per_S : REAL;
	END_STRUCT;
	Target_typ : 	STRUCT
		VBlock_Occupied : BOOL;
		VBlock_Dispensed : ARRAY[0..MAX_IDX_VALVES]OF BOOL;
	END_STRUCT;
	AS3500HS_Disp_Debug_Items_typ : 	STRUCT
		Count : DINT;
		Latch_Position : AS3500HS_Position_Var_typ;
	END_STRUCT;
	AS3500_Disp_Debug_typ : 	STRUCT
		Disp_Trigger_Count : ARRAY[0..MAX_IDX_VALVES]OF AS3500HS_Disp_Debug_Items_typ;
		Disp_Cycle_Count : ARRAY[0..MAX_IDX_VALVES]OF AS3500HS_Disp_Debug_Items_typ;
		Disp_Flag_Twice : ARRAY[0..MAX_IDX_VALVES]OF AS3500HS_Disp_Debug_Items_typ;
		Valve_Not_Rdy : ARRAY[0..MAX_IDX_VALVES]OF AS3500HS_Disp_Debug_Items_typ;
	END_STRUCT;
	AS3500HS_Stats_typ : 	STRUCT
		total_runtime : UDINT;
		runtime_h : UDINT;
		runtime_m : UDINT;
		runtime_s : UDINT;
		Total_Num_Targets : UDINT;
		VBlock_Fraction_Pos_Last_Edge : REAL;
		Debug : AS3500_Disp_Debug_typ;
		Count_PiP_Twice_Single_Targ : AS3500HS_Disp_Debug_Items_typ;
		Dispense_Discrepancy : DINT;
	END_STRUCT;
END_TYPE
```

### Global.var - not listed in the package file held
```iecst
VAR CONSTANT
	FORCEIO_ACCESS_LEVEL : UINT := 1;
	CONFIG_ACCESS_LEVEL : UINT := 2;
	RECIPE_ACCESS_LEVEL : UINT := 1;
	DEFINE_MENU_L_HIDE_TIMEOUT_MS : UDINT := 7000;
	DEFINE_MENU_R_HIDE_TIMEOUT_MS : UDINT := 7000;
	DEFINE_HMI_SPLASHSCREEN_TO_MS : UDINT := 5000;
	MAX_IDX_TOTAL_RECIPES : UINT := 100;
	DEFINE_LOGIN_TO : REAL := 600;
END_VAR
(*Insert your comment here.*)
VAR CONSTANT
	MAX_IDX_CREASES : UDINT := 19;
END_VAR
(*Insert your comment here.*)
(*Insert your comment here.*)
VAR RETAIN
	gRecCfg : Global_Par_typ;
END_VAR
VAR
	gAcknowledge : Machine_Alarms_typ;
	gAlarms : Machine_Alarms_typ;
	gMachineName : {REDUND_UNREPLICABLE} STRING[80] := 'Aries';
	gProjectDate : {REDUND_UNREPLICABLE} STRING[80] := '10. April 2017';
	gVersion : {REDUND_UNREPLICABLE} STRING[80] := 'R741';
END_VAR
(*Insert your comment here.*)
VAR
	Axis1 : ACP10AXIS_typ;
	AxisControl : MpAxisBasic;
	AxisPar : MpAxisBasicParType;
	Alarm_Feed : MpAlarmBasicUIConnect20Type := (0);
	Alarm_Feed_UI : MpAlarmBasicUI := (0);
END_VAR
(*Insert your comment here.*)
VAR
	MachineState : AriesMachineState_Enum;
	ProcessState : CreaserPrcsState_Enum;
END_VAR
(*Insert your comment here.*)
VAR
	IO : AriesIOPoints_typ;
	IO_LastCycle : AriesIOPoints_typ;
END_VAR
(*Insert your comment here.*)
VAR
	AppAlarms : MpAlarmBasicUIConnect20Type;
	AppAlarms_FBK : MpAlarmBasic;
	AppAlarms_UI : USINT;
END_VAR
(*Insert your comment here.*)
VAR RETAIN
	gStatistics : Global_Statistics_typ;
END_VAR
(*Insert your comment here.*)
VAR
	gAlarmResetRequested : BOOL;
	iMachineErrorReset : BOOL;
	iStartCommand : BOOL;
	iSoftStopCommand : BOOL;
	gSimulateMachine : BOOL;
END_VAR
(*Insert your comment here.*)
VAR CONSTANT
	DEFINE_MM_ROLLER_REV : REAL := 125.664;
END_VAR
VAR
	delta_Board_Position : REAL;
	RollerPos_LastCycle : REAL;
	RollerPos_ThisCycle : REAL;
	Current_Board_Position : REAL;
	Latch_Board_Length : REAL;
	Current_Crease_Section_Length : REAL;
END_VAR
(*Insert your comment here.*)
(*Insert your comment here.*)
```

### GlobalVariables.var - not listed in the package file held
```iecst
(*Insert your comment here.*)
(*Insert your comment here.*)
VAR RETAIN
	gRecCfg : Global_Par_typ;
END_VAR
VAR
	gAlarms : Machine_Alarms_typ;
	gMachineName : {REDUND_UNREPLICABLE} STRING[80] := 'AS3500HS';
	gProjectDate : {REDUND_UNREPLICABLE} STRING[80] := '7. March 2017';
	gVersion : {REDUND_UNREPLICABLE} STRING[80] := 'TBD';
END_VAR
(*Insert your comment here.*)
VAR
	Axis : ACP10AXIS_typ;
	AxisControl : MpAxisBasic;
	AxisPar : MpAxisBasicParType;
END_VAR
(*Insert your comment here.*)
VAR
	MachineState : AriesMachineState_Enum;
	ProcessState : CreaserPrcsState_Enum;
END_VAR
(*Insert your comment here.*)
VAR
	IO : AriesIOPoints_typ;
	IO_LastCycle : AriesIOPoints_typ;
END_VAR
(*Insert your comment here.*)
VAR RETAIN
	gStatistics : Global_Statistics_typ;
END_VAR
(*Insert your comment here.*)
(*Insert your comment here.*)
(*Insert your comment here.*)
(*Insert your comment here.*)
```

Listed in the project but not available here: Logical/doc, Logical/Libraries/wbrServices/Doc, Logical/Libraries/wbrServices/wbrServices_C_Includes, Logical/Libraries/wbrServices/wbrServices.typ, Logical/Libraries/wbrServices/wbrLogSvc/wbrLogSvc.typ, Logical/Libraries/wbrServices/wbrLogSvc/wbrLogSvc.var, Logical/Libraries/wbrServices/wbrLogSvc/wbrLogSvc.fun, Logical/Libraries/wbrServices/wbrLogSvc/wbrLogSvc.c, Logical/Libraries/wbrServices/wbrServicesGlobal.var, Logical/Libraries/wbrServices/Cyclic, Logical/Libraries/wbrServices/TimerServices, Logical/Application/Creaser/Types.typ, Logical/Application/Creaser/Action_Manage_Update_Total_Runtime.st, Logical/Application/Creaser/Action_Tally_Board_L.st, Logical/Application/Creaser/LocalFunctions.fun, Logical/Application/Creaser/PulseTrain.st, Logical/Application/Creaser/Action_Move_Photoeye_Offset.st, Logical/Application/Dispense/libValve/Variables.var, Logical/Application/Dispense/libValve/libValve.fun, Logical/Application/Dispense/libValve/Enumerations.typ, Logical/Application/Dispense/libValve/RecCfgParams.typ, Logical/Application/Dispense/libValve/AlarmsWarnings.typ, Logical/Application/Dispense/Texts/Params, Logical/HMI/Generic_Controls.typ, Logical/HMI/HMI_Pages.typ, Logical/HMI/HMIdialog.typ, Logical/HMI/HMImsgScroll.typ, Logical/HMI/HMIForceIO.typ, Logical/HMI/HMIremmem.typ, Logical/acp10etxen
